LIN {X 0,Y 285.275,Z 343.324,A -85,B 0,C 180,E1 -18502.278,E2 -18502.278} C_VEL
LIN {X 0,Y 279.28,Z 333.872,A -85,B 0,C 180,E1 -18504.288,E2 -18504.288} C_VEL
LIN {X 0,Y 273.466,Z 325.227,A -85,B 0,C 180,E1 -18506.402,E2 -18506.402} C_VEL
LIN {X 0,Y 268.524,Z 318.8,A -85,B 0,C 180,E1 -18508.326,E2 -18508.326} C_VEL
LIN {X 0,Y 265.812,Z 315.625,A -85,B 0,C 180,E1 -18509.442,E2 -18509.442} C_VEL
LIN {X 0,Y 264.728,Z 313.915,A -85,B 0,C 180,E1 -18509.928,E2 -18509.928} C_VEL
LIN {X 0,Y 262.153,Z 311.495,A -85,B 0,C 180,E1 -18511.038,E2 -18511.038} C_VEL
LIN {X 0,Y 260.63,Z 308.609,A -85,B 0,C 180,E1 -18511.807,E2 -18511.807} C_VEL
LIN {X 0,Y 258.077,Z 306.933,A -85,B 0,C 180,E1 -18512.972,E2 -18512.972} C_VEL
LIN {X 0,Y 256.551,Z 304.575,A -85,B 0,C 180,E1 -18513.786,E2 -18513.786} C_VEL
LIN {X 0,Y 256.134,Z 302.894,A -85,B 0,C 180,E1 -18514.093,E2 -18514.093} C_VEL
LIN {X 0,Y 256.099,Z 302.893,A -85,B 0,C 180,E1 -18517.407,E2 -18517.407} C_VEL
LIN {X 0,Y 256.184,Z 302.852,A -85,B 0,C 180,E1 -18520.78,E2 -18520.78} C_VEL
LIN {X 0,Y 256.293,Z 302.86,A -85,B 0,C 180,E1 -18524.085,E2 -18524.085} C_VEL
LIN {X 0,Y 256.292,Z 302.834,A -85,B 0,C 180,E1 -18527.328,E2 -18527.328} C_VEL
LIN {X 0,Y 256.514,Z 302.81,A -85,B 0,C 180,E1 -18532.127,E2 -18532.127} C_VEL
LIN {X 0,Y 256.498,Z 302.847,A -85,B 0,C 180,E1 -18536.859,E2 -18536.859} C_VEL
LIN {X 0,Y 256.756,Z 302.772,A -85,B 0,C 180,E1 -18540,E2 -18540} C_VEL
LIN {X 0,Y 256.497,Z 302.827,A -85,B 0,C 180,E1 -18543.142,E2 -18543.142} C_VEL
LIN {X 0,Y 256.514,Z 302.799,A -85,B 0,C 180,E1 -18547.874,E2 -18547.874} C_VEL
LIN {X 0,Y 256.293,Z 302.863,A -85,B 0,C 180,E1 -18552.672,E2 -18552.672} C_VEL
LIN {X 0,Y 256.26,Z 302.84,A -85,B 0,C 180,E1 -18556.286,E2 -18556.286} C_VEL
LIN {X 0,Y 256.162,Z 302.855,A -85,B 0,C 180,E1 -18560.896,E2 -18560.896} C_VEL
LIN {X 0,Y 256.17,Z 302.889,A -85,B 0,C 180,E1 -18565.13,E2 -18565.13} C_VEL
LIN {X 0,Y 256.122,Z 302.89,A -85,B 0,C 180,E1 -18566.371,E2 -18566.371} C_VEL
LIN {X 0,Y 256.849,Z 305.157,A -85,B 0,C 180,E1 -18566.839,E2 -18566.839} C_VEL
LIN {X 0,Y 258.629,Z 307.429,A -85,B 0,C 180,E1 -18567.75,E2 -18567.75} C_VEL
LIN {X 0,Y 260.674,Z 308.807,A -85,B 0,C 180,E1 -18568.678,E2 -18568.678} C_VEL
LIN {X 0,Y 262.404,Z 311.878,A -85,B 0,C 180,E1 -18569.537,E2 -18569.537} C_VEL
LIN {X 0,Y 265.164,Z 314.465,A -85,B 0,C 180,E1 -18570.717,E2 -18570.717} C_VEL
LIN {X 0,Y 267.552,Z 317.88,A -85,B 0,C 180,E1 -18571.748,E2 -18571.748} C_VEL
LIN {X 0,Y 269.408,Z 319.837,A -85,B 0,C 180,E1 -18572.481,E2 -18572.481} C_VEL
LIN {X 0,Y 272.405,Z 323.638,A -85,B 0,C 180,E1 -18573.645,E2 -18573.645} C_VEL
LIN {X 0,Y 277.071,Z 329.846,A -85,B 0,C 180,E1 -18575.356,E2 -18575.356} C_VEL
LIN {X 0,Y 282.926,Z 337.789,A -85,B 0,C 180,E1 -18577.336,E2 -18577.336} C_VEL
LIN {X 0,Y 289.288,Z 347.193,A -85,B 0,C 180,E1 -18579.335,E2 -18579.335} C_VEL
LIN {X 0,Y 297.565,Z 360.153,A -85,B 0,C 180,E1 -18581.721,E2 -18581.721} C_VEL
LIN {X 0,Y 305.62,Z 374.188,A -85,B 0,C 180,E1 -18583.871,E2 -18583.871} C_VEL
LIN {X 0,Y 306.514,Z 376.066,A -85,B 0,C 180,E1 -18584.108,E2 -18584.108} C_VEL
LIN {X 0,Y 299.995,Z 497.473,A -85,B 0,C 180,E1 -18586.903,E2 -18586.903} C_VEL
LIN {X 0,Y 298.313,Z 513.582,A -85,B 0,C 180,E1 -18587.48,E2 -18587.48} C_VEL
LIN {X 0,Y 296.185,Z 528.781,A -85,B 0,C 180,E1 -18588.251,E2 -18588.251} C_VEL
LIN {X 0,Y 293.455,Z 544.075,A -85,B 0,C 180,E1 -18589.261,E2 -18589.261} C_VEL
LIN {X 0,Y 290.548,Z 557.266,A -85,B 0,C 180,E1 -18590.359,E2 -18590.359} C_VEL
LIN {X 0,Y 286.959,Z 571.758,A -85,B 0,C 180,E1 -18591.848,E2 -18591.848} C_VEL
LIN {X 0,Y 282.878,Z 585.913,A -85,B 0,C 180,E1 -18593.618,E2 -18593.618} C_VEL
LIN {X 0,Y 278.715,Z 599.171,A -85,B 0,C 180,E1 -18595.653,E2 -18595.653} C_VEL
LIN {X 0,Y 274.546,Z 611.271,A -85,B 0,C 180,E1 -18597.916,E2 -18597.916} C_VEL
LIN {X 0,Y 270.52,Z 622.375,A -85,B 0,C 180,E1 -18600.422,E2 -18600.422} C_VEL
LIN {X 0,Y 266.38,Z 633.115,A -85,B 0,C 180,E1 -18603.352,E2 -18603.352} C_VEL
LIN {X 0,Y 263.033,Z 642.124,A -85,B 0,C 180,E1 -18606.373,E2 -18606.373} C_VEL
LIN {X 0,Y 260.17,Z 649.651,A -85,B 0,C 180,E1 -18609.441,E2 -18609.441} C_VEL
LIN {X 0,Y 257.502,Z 657.205,A -85,B 0,C 180,E1 -18613.347,E2 -18613.347} C_VEL
LIN {X 0,Y 255.967,Z 661.885,A -85,B 0,C 180,E1 -18616.504,E2 -18616.504} C_VEL
LIN {X 0,Y 255.175,Z 664.727,A -85,B 0,C 180,E1 -18618.884,E2 -18618.884} C_VEL
LIN {X 0,Y 254.496,Z 667.617,A -85,B 0,C 180,E1 -18622.063,E2 -18622.063} C_VEL
LIN {X 0,Y 254.141,Z 669.513,A -85,B 0,C 180,E1 -18625.241,E2 -18625.241} C_VEL
LIN {X 0,Y 254.078,Z 670.469,A -85,B 0,C 180,E1 -18628.415,E2 -18628.415} C_VEL
LIN {X 0,Y 254.078,Z 670.481,A -85,B 0,C 180,E1 -18631.585,E2 -18631.585} C_VEL
LIN {X 0,Y 254.141,Z 669.574,A -85,B 0,C 180,E1 -18634.759,E2 -18634.759} C_VEL
LIN {X 0,Y 254.494,Z 667.702,A -85,B 0,C 180,E1 -18637.936,E2 -18637.936} C_VEL
LIN {X 0,Y 255.145,Z 664.86,A -85,B 0,C 180,E1 -18641.117,E2 -18641.117} C_VEL
LIN {X 0,Y 256.293,Z 660.99,A -85,B 0,C 180,E1 -18644.288,E2 -18644.288} C_VEL
LIN {X 0,Y 258.026,Z 655.765,A -85,B 0,C 180,E1 -18647.576,E2 -18647.576} C_VEL
LIN {X 0,Y 260.127,Z 649.916,A -85,B 0,C 180,E1 -18650.562,E2 -18650.562} C_VEL
LIN {X 0,Y 263.41,Z 641.424,A -85,B 0,C 180,E1 -18654.009,E2 -18654.009} C_VEL
LIN {X 0,Y 266.775,Z 632.258,A -85,B 0,C 180,E1 -18657.029,E2 -18657.029} C_VEL
LIN {X 0,Y 270.404,Z 622.812,A -85,B 0,C 180,E1 -18659.592,E2 -18659.592} C_VEL
LIN {X 0,Y 274.457,Z 611.863,A -85,B 0,C 180,E1 -18662.079,E2 -18662.079} C_VEL
LIN {X 0,Y 278.265,Z 600.716,A -85,B 0,C 180,E1 -18664.191,E2 -18664.191} C_VEL
LIN {X 0,Y 282.046,Z 588.931,A -85,B 0,C 180,E1 -18666.063,E2 -18666.063} C_VEL
LIN {X 0,Y 285.784,Z 576.531,A -85,B 0,C 180,E1 -18667.714,E2 -18667.714} C_VEL
LIN {X 0,Y 289.199,Z 563.238,A -85,B 0,C 180,E1 -18669.186,E2 -18669.186} C_VEL
LIN {X 0,Y 292.454,Z 549.191,A -85,B 0,C 180,E1 -18670.454,E2 -18670.454} C_VEL
LIN {X 0,Y 295.442,Z 534.168,A -85,B 0,C 180,E1 -18671.536,E2 -18671.536} C_VEL
LIN {X 0,Y 297.702,Z 518.897,A -85,B 0,C 180,E1 -18672.398,E2 -18672.398} C_VEL
LIN {X 0,Y 299.684,Z 502.058,A -85,B 0,C 180,E1 -18673.063,E2 -18673.063} C_VEL
LIN {X 0,Y 301.058,Z 481.051,A -85,B 0,C 180,E1 -18673.617,E2 -18673.617} C_VEL
LIN {X 0,Y 306.585,Z 376.776,A -85,B 0,C 180,E1 -18675.989,E2 -18675.989} C_VEL
LIN {X 0,Y 306.295,Z 375.437,A -85,B 0,C 180,E1 -18676.09,E2 -18676.09} C_VEL
LIN {X 0,Y 299.197,Z 362.765,A -85,B 0,C 180,E1 -18677.975,E2 -18677.975} C_VEL
LIN {X 0,Y 291.683,Z 350.766,A -85,B 0,C 180,E1 -18680.102,E2 -18680.102} C_VEL
LIN {X 0,Y 287.132,Z 343.847,A -85,B 0,C 180,E1 -18681.48,E2 -18681.48} C_VEL
LIN {X 0,Y 284.356,Z 340.758,A -85,B 0,C 180,E1 -18682.318,E2 -18682.318} C_VEL
LIN {X 0,Y 279.14,Z 337.36,A -85,B 0,C 180,E1 -18683.882,E2 -18683.882} C_VEL
LIN {X 0,Y 273.02,Z 333.547,A -85,B 0,C 180,E1 -18685.87,E2 -18685.87} C_VEL
LIN {X 0,Y 271.247,Z 331.735,A -85,B 0,C 180,E1 -18686.516,E2 -18686.516} C_VEL
LIN {X 0,Y 269.262,Z 329.124,A -85,B 0,C 180,E1 -18687.291,E2 -18687.291} C_VEL
LIN {X 0,Y 265.972,Z 324.859,A -85,B 0,C 180,E1 -18688.637,E2 -18688.637} C_VEL
LIN {X 0,Y 263.083,Z 321.248,A -85,B 0,C 180,E1 -18689.886,E2 -18689.886} C_VEL
LIN {X 0,Y 262.021,Z 319.981,A -85,B 0,C 180,E1 -18690.361,E2 -18690.361} C_VEL
LIN {X 0,Y 259.368,Z 316.979,A -85,B 0,C 180,E1 -18691.587,E2 -18691.587} C_VEL
LIN {X 0,Y 258.32,Z 315.094,A -85,B 0,C 180,E1 -18692.134,E2 -18692.134} C_VEL
LIN {X 0,Y 255.6,Z 312.813,A -85,B 0,C 180,E1 -18693.46,E2 -18693.46} C_VEL
LIN {X 0,Y 253.93,Z 309.833,A -85,B 0,C 180,E1 -18694.423,E2 -18694.423} C_VEL
LIN {X 0,Y 250.638,Z 307.386,A -85,B 0,C 180,E1 -18696.229,E2 -18696.229} C_VEL
LIN {X 0,Y 249.411,Z 305.23,A -85,B 0,C 180,E1 -18697.039,E2 -18697.039} C_VEL
LIN {X 0,Y 249.069,Z 303.741,A -85,B 0,C 180,E1 -18697.39,E2 -18697.39} C_VEL
LIN {X 0,Y 249.135,Z 303.748,A -85,B 0,C 180,E1 -18701.922,E2 -18701.922} C_VEL
LIN {X 0,Y 249.196,Z 303.728,A -85,B 0,C 180,E1 -18705.296,E2 -18705.296} C_VEL
LIN {X 0,Y 249.423,Z 303.689,A -85,B 0,C 180,E1 -18710.465,E2 -18710.465} C_VEL
LIN {X 0,Y 249.46,Z 303.724,A -85,B 0,C 180,E1 -18713.529,E2 -18713.529} C_VEL
LIN {X 0,Y 249.674,Z 303.664,A -85,B 0,C 180,E1 -18718.387,E2 -18718.387} C_VEL
LIN {X 0,Y 249.674,Z 303.684,A -85,B 0,C 180,E1 -18721.613,E2 -18721.613} C_VEL
LIN {X 0,Y 249.46,Z 303.713,A -85,B 0,C 180,E1 -18726.47,E2 -18726.47} C_VEL
LIN {X 0,Y 249.387,Z 303.699,A -85,B 0,C 180,E1 -18729.734,E2 -18729.734} C_VEL
LIN {X 0,Y 249.204,Z 303.75,A -85,B 0,C 180,E1 -18734.703,E2 -18734.703} C_VEL
LIN {X 0,Y 249.138,Z 303.758,A -85,B 0,C 180,E1 -18738.077,E2 -18738.077} C_VEL
LIN {X 0,Y 249.053,Z 303.773,A -85,B 0,C 180,E1 -18742.283,E2 -18742.283} C_VEL
LIN {X 0,Y 249.862,Z 306.296,A -85,B 0,C 180,E1 -18742.916,E2 -18742.916} C_VEL
LIN {X 0,Y 251.817,Z 308.516,A -85,B 0,C 180,E1 -18744.09,E2 -18744.09} C_VEL
LIN {X 0,Y 253.91,Z 309.796,A -85,B 0,C 180,E1 -18745.199,E2 -18745.199} C_VEL
LIN {X 0,Y 255.481,Z 312.696,A -85,B 0,C 180,E1 -18746.113,E2 -18746.113} C_VEL
LIN {X 0,Y 258.017,Z 314.954,A -85,B 0,C 180,E1 -18747.364,E2 -18747.364} C_VEL
LIN {X 0,Y 258.576,Z 315.522,A -85,B 0,C 180,E1 -18747.634,E2 -18747.634} C_VEL
LIN {X 0,Y 260.685,Z 318.703,A -85,B 0,C 180,E1 -18748.678,E2 -18748.678} C_VEL
LIN {X 0,Y 262.953,Z 321.044,A -85,B 0,C 180,E1 -18749.688,E2 -18749.688} C_VEL
LIN {X 0,Y 265.557,Z 324.493,A -85,B 0,C 180,E1 -18750.83,E2 -18750.83} C_VEL
LIN {X 0,Y 267.011,Z 326.216,A -85,B 0,C 180,E1 -18751.432,E2 -18751.432} C_VEL
LIN {X 0,Y 271.996,Z 332.99,A -85,B 0,C 180,E1 -18753.417,E2 -18753.417} C_VEL
LIN {X 0,Y 278.858,Z 343.518,A -85,B 0,C 180,E1 -18755.936,E2 -18755.936} C_VEL
LIN {X 0,Y 286.061,Z 355.576,A -85,B 0,C 180,E1 -18758.347,E2 -18758.347} C_VEL
LIN {X 0,Y 293.093,Z 368.397,A -85,B 0,C 180,E1 -18760.517,E2 -18760.517} C_VEL
LIN {X 0,Y 299.812,Z 382.28,A -85,B 0,C 180,E1 -18762.471,E2 -18762.471} C_VEL
LIN {X 0,Y 301.353,Z 385.582,A -85,B 0,C 180,E1 -18762.901,E2 -18762.901} C_VEL
LIN {X 0,Y 294.372,Z 510.514,A -85,B 0,C 180,E1 -18765.799,E2 -18765.799} C_VEL
LIN {X 0,Y 292.365,Z 527.573,A -85,B 0,C 180,E1 -18766.402,E2 -18766.402} C_VEL
LIN {X 0,Y 289.707,Z 543.728,A -85,B 0,C 180,E1 -18767.215,E2 -18767.215} C_VEL
LIN {X 0,Y 286.53,Z 559.561,A -85,B 0,C 180,E1 -18768.294,E2 -18768.294} C_VEL
LIN {X 0,Y 283.015,Z 574.179,A -85,B 0,C 180,E1 -18769.553,E2 -18769.553} C_VEL
LIN {X 0,Y 278.905,Z 588.943,A -85,B 0,C 180,E1 -18771.143,E2 -18771.143} C_VEL
LIN {X 0,Y 274.506,Z 602.929,A -85,B 0,C 180,E1 -18773.012,E2 -18773.012} C_VEL
LIN {X 0,Y 270.049,Z 615.655,A -85,B 0,C 180,E1 -18775.072,E2 -18775.072} C_VEL
LIN {X 0,Y 265.467,Z 628.288,A -85,B 0,C 180,E1 -18777.582,E2 -18777.582} C_VEL
LIN {X 0,Y 261.478,Z 639.066,A -85,B 0,C 180,E1 -18780.183,E2 -18780.183} C_VEL
LIN {X 0,Y 257.372,Z 649.469,A -85,B 0,C 180,E1 -18783.221,E2 -18783.221} C_VEL
LIN {X 0,Y 254.04,Z 658.16,A -85,B 0,C 180,E1 -18786.351,E2 -18786.351} C_VEL
LIN {X 0,Y 251.411,Z 665.441,A -85,B 0,C 180,E1 -18789.548,E2 -18789.548} C_VEL
LIN {X 0,Y 249.437,Z 671.625,A -85,B 0,C 180,E1 -18792.877,E2 -18792.877} C_VEL
LIN {X 0,Y 247.855,Z 677.362,A -85,B 0,C 180,E1 -18796.889,E2 -18796.889} C_VEL
LIN {X 0,Y 247.105,Z 680.799,A -85,B 0,C 180,E1 -18800.175,E2 -18800.175} C_VEL
LIN {X 0,Y 246.858,Z 683.304,A -85,B 0,C 180,E1 -18803.461,E2 -18803.461} C_VEL
LIN {X 0,Y 246.852,Z 684.721,A -85,B 0,C 180,E1 -18806.736,E2 -18806.736} C_VEL
LIN {X 0,Y 246.981,Z 685.254,A -85,B 0,C 180,E1 -18810,E2 -18810} C_VEL
LIN {X 0,Y 246.852,Z 684.711,A -85,B 0,C 180,E1 -18813.264,E2 -18813.264} C_VEL
LIN {X 0,Y 246.859,Z 683.284,A -85,B 0,C 180,E1 -18816.539,E2 -18816.539} C_VEL
LIN {X 0,Y 247.105,Z 680.77,A -85,B 0,C 180,E1 -18819.825,E2 -18819.825} C_VEL
LIN {X 0,Y 248.115,Z 676.241,A -85,B 0,C 180,E1 -18823.932,E2 -18823.932} C_VEL
LIN {X 0,Y 249.436,Z 671.576,A -85,B 0,C 180,E1 -18827.124,E2 -18827.124} C_VEL
LIN {X 0,Y 252.01,Z 663.718,A -85,B 0,C 180,E1 -18831.256,E2 -18831.256} C_VEL
LIN {X 0,Y 254.904,Z 655.834,A -85,B 0,C 180,E1 -18834.517,E2 -18834.517} C_VEL
LIN {X 0,Y 258.342,Z 646.883,A -85,B 0,C 180,E1 -18837.547,E2 -18837.547} C_VEL
LIN {X 0,Y 262.56,Z 635.997,A -85,B 0,C 180,E1 -18840.569,E2 -18840.569} C_VEL
LIN {X 0,Y 266.111,Z 626.507,A -85,B 0,C 180,E1 -18842.779,E2 -18842.779} C_VEL
LIN {X 0,Y 270.039,Z 615.479,A -85,B 0,C 180,E1 -18844.929,E2 -18844.929} C_VEL
LIN {X 0,Y 274.491,Z 602.717,A -85,B 0,C 180,E1 -18846.991,E2 -18846.991} C_VEL
LIN {X 0,Y 278.509,Z 589.956,A -85,B 0,C 180,E1 -18848.709,E2 -18848.709} C_VEL
LIN {X 0,Y 282.572,Z 575.469,A -85,B 0,C 180,E1 -18850.29,E2 -18850.29} C_VEL
LIN {X 0,Y 286.078,Z 561.175,A -85,B 0,C 180,E1 -18851.552,E2 -18851.552} C_VEL
LIN {X 0,Y 289.237,Z 545.847,A -85,B 0,C 180,E1 -18852.634,E2 -18852.634} C_VEL
LIN {X 0,Y 292.012,Z 529.58,A -85,B 0,C 180,E1 -18853.486,E2 -18853.486} C_VEL
LIN {X 0,Y 294.055,Z 512.875,A -85,B 0,C 180,E1 -18854.098,E2 -18854.098} C_VEL
LIN {X 0,Y 295.614,Z 486.575,A -85,B 0,C 180,E1 -18854.773,E2 -18854.773} C_VEL
LIN {X 0,Y 301.244,Z 385.521,A -85,B 0,C 180,E1 -18857.076,E2 -18857.076} C_VEL
LIN {X 0,Y 294.208,Z 370.745,A -85,B 0,C 180,E1 -18859.093,E2 -18859.093} C_VEL
LIN {X 0,Y 287.651,Z 358.497,A -85,B 0,C 180,E1 -18861.084,E2 -18861.084} C_VEL
LIN {X 0,Y 280.685,Z 346.559,A -85,B 0,C 180,E1 -18863.361,E2 -18863.361} C_VEL
LIN {X 0,Y 275.917,Z 339.051,A -85,B 0,C 180,E1 -18865.033,E2 -18865.033} C_VEL
LIN {X 0,Y 270.151,Z 330.37,A -85,B 0,C 180,E1 -18867.219,E2 -18867.219} C_VEL
LIN {X 0,Y 265.908,Z 324.844,A -85,B 0,C 180,E1 -18868.934,E2 -18868.934} C_VEL
LIN {X 0,Y 263.062,Z 321.269,A -85,B 0,C 180,E1 -18870.16,E2 -18870.16} C_VEL
LIN {X 0,Y 261.902,Z 319.861,A -85,B 0,C 180,E1 -18870.678,E2 -18870.678} C_VEL
LIN {X 0,Y 259.328,Z 316.934,A -85,B 0,C 180,E1 -18871.864,E2 -18871.864} C_VEL
LIN {X 0,Y 258.206,Z 315.058,A -85,B 0,C 180,E1 -18872.438,E2 -18872.438} C_VEL
LIN {X 0,Y 255.549,Z 312.778,A -85,B 0,C 180,E1 -18873.73,E2 -18873.73} C_VEL
LIN {X 0,Y 253.879,Z 309.778,A -85,B 0,C 180,E1 -18874.689,E2 -18874.689} C_VEL
LIN {X 0,Y 250.643,Z 307.395,A -85,B 0,C 180,E1 -18876.449,E2 -18876.449} C_VEL
LIN {X 0,Y 249.403,Z 305.259,A -85,B 0,C 180,E1 -18877.258,E2 -18877.258} C_VEL
LIN {X 0,Y 249.052,Z 303.764,A -85,B 0,C 180,E1 -18877.607,E2 -18877.607} C_VEL
LIN {X 0,Y 249.138,Z 303.743,A -85,B 0,C 180,E1 -18881.923,E2 -18881.923} C_VEL
LIN {X 0,Y 249.199,Z 303.721,A -85,B 0,C 180,E1 -18885.297,E2 -18885.297} C_VEL
LIN {X 0,Y 249.386,Z 303.729,A -85,B 0,C 180,E1 -18890.517,E2 -18890.517} C_VEL
LIN {X 0,Y 249.452,Z 303.679,A -85,B 0,C 180,E1 -18893.53,E2 -18893.53} C_VEL
LIN {X 0,Y 249.675,Z 303.678,A -85,B 0,C 180,E1 -18898.387,E2 -18898.387} C_VEL
LIN {X 0,Y 249.674,Z 303.653,A -85,B 0,C 180,E1 -18901.613,E2 -18901.613} C_VEL
LIN {X 0,Y 249.44,Z 303.689,A -85,B 0,C 180,E1 -18906.711,E2 -18906.711} C_VEL
LIN {X 0,Y 249.342,Z 303.703,A -85,B 0,C 180,E1 -18909.737,E2 -18909.737} C_VEL
LIN {X 0,Y 249.196,Z 303.715,A -85,B 0,C 180,E1 -18914.704,E2 -18914.704} C_VEL
LIN {X 0,Y 249.135,Z 303.759,A -85,B 0,C 180,E1 -18918.078,E2 -18918.078} C_VEL
LIN {X 0,Y 249.037,Z 303.739,A -85,B 0,C 180,E1 -18922.395,E2 -18922.395} C_VEL
LIN {X 0,Y 249.035,Z 303.765,A -85,B 0,C 180,E1 -18922.888,E2 -18922.888} C_VEL
LIN {X 0,Y 249.722,Z 306.013,A -85,B 0,C 180,E1 -18923.424,E2 -18923.424} C_VEL
LIN {X 0,Y 251.586,Z 308.326,A -85,B 0,C 180,E1 -18924.553,E2 -18924.553} C_VEL
LIN {X 0,Y 253.921,Z 309.828,A -85,B 0,C 180,E1 -18925.79,E2 -18925.79} C_VEL
LIN {X 0,Y 255.614,Z 312.839,A -85,B 0,C 180,E1 -18926.758,E2 -18926.758} C_VEL
LIN {X 0,Y 258.488,Z 315.485,A -85,B 0,C 180,E1 -18928.161,E2 -18928.161} C_VEL
LIN {X 0,Y 260.8,Z 318.863,A -85,B 0,C 180,E1 -18929.293,E2 -18929.293} C_VEL
LIN {X 0,Y 262.853,Z 320.924,A -85,B 0,C 180,E1 -18930.199,E2 -18930.199} C_VEL
LIN {X 0,Y 265.628,Z 324.576,A -85,B 0,C 180,E1 -18931.408,E2 -18931.408} C_VEL
LIN {X 0,Y 267.03,Z 326.203,A -85,B 0,C 180,E1 -18931.984,E2 -18931.984} C_VEL
LIN {X 0,Y 270.974,Z 331.365,A -85,B 0,C 180,E1 -18933.551,E2 -18933.551} C_VEL
LIN {X 0,Y 277.003,Z 339.459,A -85,B 0,C 180,E1 -18935.758,E2 -18935.758} C_VEL
LIN {X 0,Y 284.758,Z 350.731,A -85,B 0,C 180,E1 -18938.342,E2 -18938.342} C_VEL
LIN {X 0,Y 293.587,Z 364.766,A -85,B 0,C 180,E1 -18941.005,E2 -18941.005} C_VEL
LIN {X 0,Y 301.429,Z 378.591,A -85,B 0,C 180,E1 -18943.18,E2 -18943.18} C_VEL
LIN {X 0,Y 294.933,Z 496.966,A -85,B 0,C 180,E1 -18945.947,E2 -18945.947} C_VEL
LIN {X 0,Y 293.248,Z 512.887,A -85,B 0,C 180,E1 -18946.507,E2 -18946.507} C_VEL
LIN {X 0,Y 290.915,Z 528.997,A -85,B 0,C 180,E1 -18947.317,E2 -18947.317} C_VEL
LIN {X 0,Y 288.115,Z 544.289,A -85,B 0,C 180,E1 -18948.34,E2 -18948.34} C_VEL
LIN {X 0,Y 285.105,Z 557.479,A -85,B 0,C 180,E1 -18949.447,E2 -18949.447} C_VEL
LIN {X 0,Y 281.748,Z 570.559,A -85,B 0,C 180,E1 -18950.782,E2 -18950.782} C_VEL
LIN {X 0,Y 277.6,Z 584.956,A -85,B 0,C 180,E1 -18952.584,E2 -18952.584} C_VEL
LIN {X 0,Y 273.574,Z 597.276,A -85,B 0,C 180,E1 -18954.463,E2 -18954.463} C_VEL
LIN {X 0,Y 269.106,Z 609.715,A -85,B 0,C 180,E1 -18956.74,E2 -18956.74} C_VEL
LIN {X 0,Y 264.892,Z 621.112,A -85,B 0,C 180,E1 -18959.288,E2 -18959.288} C_VEL
LIN {X 0,Y 260.996,Z 630.875,A -85,B 0,C 180,E1 -18961.886,E2 -18961.886} C_VEL
LIN {X 0,Y 257.317,Z 640.237,A -85,B 0,C 180,E1 -18964.954,E2 -18964.954} C_VEL
LIN {X 0,Y 254.161,Z 648.073,A -85,B 0,C 180,E1 -18968.081,E2 -18968.081} C_VEL
LIN {X 0,Y 251.668,Z 654.605,A -85,B 0,C 180,E1 -18971.268,E2 -18971.268} C_VEL
LIN {X 0,Y 249.772,Z 659.884,A -85,B 0,C 180,E1 -18974.496,E2 -18974.496} C_VEL
LIN {X 0,Y 248.656,Z 663.146,A -85,B 0,C 180,E1 -18976.932,E2 -18976.932} C_VEL
LIN {X 0,Y 247.763,Z 666.493,A -85,B 0,C 180,E1 -18980.201,E2 -18980.201} C_VEL
LIN {X 0,Y 247.196,Z 668.926,A -85,B 0,C 180,E1 -18983.47,E2 -18983.47} C_VEL
LIN {X 0,Y 247.015,Z 670.301,A -85,B 0,C 180,E1 -18986.738,E2 -18986.738} C_VEL
LIN {X 0,Y 246.99,Z 670.831,A -85,B 0,C 180,E1 -18990,E2 -18990} C_VEL
LIN {X 0,Y 247.014,Z 670.338,A -85,B 0,C 180,E1 -18993.262,E2 -18993.262} C_VEL
LIN {X 0,Y 247.195,Z 668.997,A -85,B 0,C 180,E1 -18996.53,E2 -18996.53} C_VEL
LIN {X 0,Y 247.755,Z 666.601,A -85,B 0,C 180,E1 -18999.799,E2 -18999.799} C_VEL
LIN {X 0,Y 248.626,Z 663.298,A -85,B 0,C 180,E1 -19003.07,E2 -19003.07} C_VEL
LIN {X 0,Y 250.608,Z 657.647,A -85,B 0,C 180,E1 -19007.101,E2 -19007.101} C_VEL
LIN {X 0,Y 253.413,Z 650.124,A -85,B 0,C 180,E1 -19011.133,E2 -19011.133} C_VEL
LIN {X 0,Y 256.874,Z 641.632,A -85,B 0,C 180,E1 -19014.66,E2 -19014.66} C_VEL
LIN {X 0,Y 260.406,Z 632.465,A -85,B 0,C 180,E1 -19017.746,E2 -19017.746} C_VEL
LIN {X 0,Y 264.196,Z 623.019,A -85,B 0,C 180,E1 -19020.359,E2 -19020.359} C_VEL
LIN {X 0,Y 268.123,Z 612.898,A -85,B 0,C 180,E1 -19022.719,E2 -19022.719} C_VEL
LIN {X 0,Y 272.379,Z 600.922,A -85,B 0,C 180,E1 -19025.036,E2 -19025.036} C_VEL
LIN {X 0,Y 276.343,Z 589.134,A -85,B 0,C 180,E1 -19026.929,E2 -19026.929} C_VEL
LIN {X 0,Y 280.173,Z 576.735,A -85,B 0,C 180,E1 -19028.607,E2 -19028.607} C_VEL
LIN {X 0,Y 283.72,Z 563.441,A -85,B 0,C 180,E1 -19030.093,E2 -19030.093} C_VEL
LIN {X 0,Y 287.104,Z 549.391,A -85,B 0,C 180,E1 -19031.37,E2 -19031.37} C_VEL
LIN {X 0,Y 290.16,Z 534.367,A -85,B 0,C 180,E1 -19032.466,E2 -19032.466} C_VEL
LIN {X 0,Y 292.513,Z 519.094,A -85,B 0,C 180,E1 -19033.334,E2 -19033.334} C_VEL
LIN {X 0,Y 294.523,Z 502.501,A -85,B 0,C 180,E1 -19033.996,E2 -19033.996} C_VEL
LIN {X 0,Y 295.987,Z 480.767,A -85,B 0,C 180,E1 -19034.575,E2 -19034.575} C_VEL
LIN {X 0,Y 301.593,Z 379.214,A -85,B 0,C 180,E1 -19036.903,E2 -19036.903} C_VEL
LIN {X 0,Y 300.741,Z 377.174,A -85,B 0,C 180,E1 -19037.148,E2 -19037.148} C_VEL
LIN {X 0,Y 292.638,Z 363.121,A -85,B 0,C 180,E1 -19039.417,E2 -19039.417} C_VEL
LIN {X 0,Y 283.622,Z 348.999,A -85,B 0,C 180,E1 -19042.176,E2 -19042.176} C_VEL
LIN {X 0,Y 276.328,Z 338.452,A -85,B 0,C 180,E1 -19044.647,E2 -19044.647} C_VEL
LIN {X 0,Y 271.247,Z 331.735,A -85,B 0,C 180,E1 -19046.516,E2 -19046.516} C_VEL
LIN {X 0,Y 268.561,Z 329.352,A -85,B 0,C 180,E1 -19047.515,E2 -19047.515} C_VEL
LIN {X 0,Y 263.721,Z 327.214,A -85,B 0,C 180,E1 -19049.331,E2 -19049.331} C_VEL
LIN {X 0,Y 259.146,Z 325.104,A -85,B 0,C 180,E1 -19051.214,E2 -19051.214} C_VEL
LIN {X 0,Y 256.843,Z 322.762,A -85,B 0,C 180,E1 -19052.31,E2 -19052.31} C_VEL
LIN {X 0,Y 255.802,Z 321.309,A -85,B 0,C 180,E1 -19052.849,E2 -19052.849} C_VEL
LIN {X 0,Y 253.145,Z 318.616,A -85,B 0,C 180,E1 -19054.229,E2 -19054.229} C_VEL
LIN {X 0,Y 251.679,Z 316.151,A -85,B 0,C 180,E1 -19055.099,E2 -19055.099} C_VEL
LIN {X 0,Y 248.857,Z 313.93,A -85,B 0,C 180,E1 -19056.71,E2 -19056.71} C_VEL
LIN {X 0,Y 247.239,Z 311.109,A -85,B 0,C 180,E1 -19057.819,E2 -19057.819} C_VEL
LIN {X 0,Y 246.9,Z 310.49,A -85,B 0,C 180,E1 -19058.062,E2 -19058.062} C_VEL
LIN {X 0,Y 244.122,Z 308.824,A -85,B 0,C 180,E1 -19059.899,E2 -19059.899} C_VEL
LIN {X 0,Y 242.516,Z 306.416,A -85,B 0,C 180,E1 -19061.192,E2 -19061.192} C_VEL
LIN {X 0,Y 242.074,Z 304.631,A -85,B 0,C 180,E1 -19061.705,E2 -19061.705} C_VEL
LIN {X 0,Y 242.155,Z 304.6,A -85,B 0,C 180,E1 -19064.858,E2 -19064.858} C_VEL
LIN {X 0,Y 242.364,Z 304.568,A -85,B 0,C 180,E1 -19070.371,E2 -19070.371} C_VEL
LIN {X 0,Y 242.432,Z 304.596,A -85,B 0,C 180,E1 -19073.341,E2 -19073.341} C_VEL
LIN {X 0,Y 242.634,Z 304.539,A -85,B 0,C 180,E1 -19078.34,E2 -19078.34} C_VEL
LIN {X 0,Y 242.635,Z 304.558,A -85,B 0,C 180,E1 -19081.66,E2 -19081.66} C_VEL
LIN {X 0,Y 242.432,Z 304.592,A -85,B 0,C 180,E1 -19086.659,E2 -19086.659} C_VEL
LIN {X 0,Y 242.313,Z 304.578,A -85,B 0,C 180,E1 -19090.022,E2 -19090.022} C_VEL
LIN {X 0,Y 242.165,Z 304.625,A -85,B 0,C 180,E1 -19095.141,E2 -19095.141} C_VEL
LIN {X 0,Y 242.129,Z 304.78,A -85,B 0,C 180,E1 -19098.017,E2 -19098.017} C_VEL
LIN {X 0,Y 242.727,Z 306.822,A -85,B 0,C 180,E1 -19098.626,E2 -19098.626} C_VEL
LIN {X 0,Y 244.301,Z 308.998,A -85,B 0,C 180,E1 -19099.866,E2 -19099.866} C_VEL
LIN {X 0,Y 247.087,Z 310.745,A -85,B 0,C 180,E1 -19101.701,E2 -19101.701} C_VEL
LIN {X 0,Y 248.601,Z 313.641,A -85,B 0,C 180,E1 -19102.764,E2 -19102.764} C_VEL
LIN {X 0,Y 251.002,Z 315.788,A -85,B 0,C 180,E1 -19104.173,E2 -19104.173} C_VEL
LIN {X 0,Y 251.924,Z 316.542,A -85,B 0,C 180,E1 -19104.682,E2 -19104.682} C_VEL
LIN {X 0,Y 254.097,Z 319.804,A -85,B 0,C 180,E1 -19105.925,E2 -19105.925} C_VEL
LIN {X 0,Y 256.437,Z 322.017,A -85,B 0,C 180,E1 -19107.105,E2 -19107.105} C_VEL
LIN {X 0,Y 259.001,Z 325.572,A -85,B 0,C 180,E1 -19108.387,E2 -19108.387} C_VEL
LIN {X 0,Y 260.555,Z 327.248,A -85,B 0,C 180,E1 -19109.101,E2 -19109.101} C_VEL
LIN {X 0,Y 263.742,Z 331.281,A -85,B 0,C 180,E1 -19110.525,E2 -19110.525} C_VEL
LIN {X 0,Y 269.115,Z 338.679,A -85,B 0,C 180,E1 -19112.756,E2 -19112.756} C_VEL
LIN {X 0,Y 275.643,Z 348.883,A -85,B 0,C 180,E1 -19115.247,E2 -19115.247} C_VEL
LIN {X 0,Y 282.45,Z 360.484,A -85,B 0,C 180,E1 -19117.618,E2 -19117.618} C_VEL
LIN {X 0,Y 289.599,Z 373.783,A -85,B 0,C 180,E1 -19119.91,E2 -19119.91} C_VEL
LIN {X 0,Y 296.012,Z 387.458,A -85,B 0,C 180,E1 -19121.85,E2 -19121.85} C_VEL
LIN {X 0,Y 296.357,Z 388.202,A -85,B 0,C 180,E1 -19121.951,E2 -19121.951} C_VEL
LIN {X 0,Y 292.743,Z 450.63,A -85,B 0,C 180,E1 -19123.385,E2 -19123.385} C_VEL
LIN {X 0,Y 289.263,Z 510.944,A -85,B 0,C 180,E1 -19124.836,E2 -19124.836} C_VEL
LIN {X 0,Y 287.134,Z 528.294,A -85,B 0,C 180,E1 -19125.461,E2 -19125.461} C_VEL
LIN {X 0,Y 284.524,Z 543.528,A -85,B 0,C 180,E1 -19126.242,E2 -19126.242} C_VEL
LIN {X 0,Y 281.248,Z 559.359,A -85,B 0,C 180,E1 -19127.327,E2 -19127.327} C_VEL
LIN {X 0,Y 277.611,Z 573.975,A -85,B 0,C 180,E1 -19128.595,E2 -19128.595} C_VEL
LIN {X 0,Y 273.298,Z 588.988,A -85,B 0,C 180,E1 -19130.232,E2 -19130.232} C_VEL
LIN {X 0,Y 268.828,Z 602.724,A -85,B 0,C 180,E1 -19132.095,E2 -19132.095} C_VEL
LIN {X 0,Y 264.196,Z 615.448,A -85,B 0,C 180,E1 -19134.181,E2 -19134.181} C_VEL
LIN {X 0,Y 259.431,Z 628.081,A -85,B 0,C 180,E1 -19136.731,E2 -19136.731} C_VEL
LIN {X 0,Y 255.26,Z 638.858,A -85,B 0,C 180,E1 -19139.379,E2 -19139.379} C_VEL
LIN {X 0,Y 250.966,Z 649.261,A -85,B 0,C 180,E1 -19142.48,E2 -19142.48} C_VEL
LIN {X 0,Y 247.354,Z 658.157,A -85,B 0,C 180,E1 -19145.762,E2 -19145.762} C_VEL
LIN {X 0,Y 244.67,Z 665.232,A -85,B 0,C 180,E1 -19148.958,E2 -19148.958} C_VEL
LIN {X 0,Y 242.582,Z 671.282,A -85,B 0,C 180,E1 -19152.29,E2 -19152.29} C_VEL
LIN {X 0,Y 240.874,Z 677.154,A -85,B 0,C 180,E1 -19156.502,E2 -19156.502} C_VEL
LIN {X 0,Y 240.041,Z 680.59,A -85,B 0,C 180,E1 -19159.883,E2 -19159.883} C_VEL
LIN {X 0,Y 239.77,Z 683.096,A -85,B 0,C 180,E1 -19163.267,E2 -19163.267} C_VEL
LIN {X 0,Y 239.758,Z 684.513,A -85,B 0,C 180,E1 -19166.639,E2 -19166.639} C_VEL
LIN {X 0,Y 239.89,Z 685.047,A -85,B 0,C 180,E1 -19170,E2 -19170} C_VEL
LIN {X 0,Y 239.758,Z 684.503,A -85,B 0,C 180,E1 -19173.361,E2 -19173.361} C_VEL
LIN {X 0,Y 239.77,Z 683.075,A -85,B 0,C 180,E1 -19176.733,E2 -19176.733} C_VEL
LIN {X 0,Y 240.041,Z 680.56,A -85,B 0,C 180,E1 -19180.118,E2 -19180.118} C_VEL
LIN {X 0,Y 240.87,Z 677.113,A -85,B 0,C 180,E1 -19183.498,E2 -19183.498} C_VEL
LIN {X 0,Y 242.58,Z 671.228,A -85,B 0,C 180,E1 -19187.71,E2 -19187.71} C_VEL
LIN {X 0,Y 245.315,Z 663.506,A -85,B 0,C 180,E1 -19191.866,E2 -19191.866} C_VEL
LIN {X 0,Y 248.718,Z 654.809,A -85,B 0,C 180,E1 -19195.526,E2 -19195.526} C_VEL
LIN {X 0,Y 252.493,Z 645.429,A -85,B 0,C 180,E1 -19198.695,E2 -19198.695} C_VEL
LIN {X 0,Y 256.372,Z 635.784,A -85,B 0,C 180,E1 -19201.389,E2 -19201.389} C_VEL
LIN {X 0,Y 260.087,Z 626.294,A -85,B 0,C 180,E1 -19203.638,E2 -19203.638} C_VEL
LIN {X 0,Y 264.193,Z 615.267,A -85,B 0,C 180,E1 -19205.82,E2 -19205.82} C_VEL
LIN {X 0,Y 268.41,Z 603.682,A -85,B 0,C 180,E1 -19207.737,E2 -19207.737} C_VEL
LIN {X 0,Y 272.476,Z 591.235,A -85,B 0,C 180,E1 -19209.457,E2 -19209.457} C_VEL
LIN {X 0,Y 276.706,Z 576.843,A -85,B 0,C 180,E1 -19211.086,E2 -19211.086} C_VEL
LIN {X 0,Y 280.797,Z 560.962,A -85,B 0,C 180,E1 -19212.514,E2 -19212.514} C_VEL
LIN {X 0,Y 284.043,Z 545.632,A -85,B 0,C 180,E1 -19213.606,E2 -19213.606} C_VEL
LIN {X 0,Y 286.884,Z 529.503,A -85,B 0,C 180,E1 -19214.454,E2 -19214.454} C_VEL
LIN {X 0,Y 288.897,Z 513.718,A -85,B 0,C 180,E1 -19215.04,E2 -19215.04} C_VEL
LIN {X 0,Y 290.337,Z 491.726,A -85,B 0,C 180,E1 -19215.629,E2 -19215.629} C_VEL
LIN {X 0,Y 296.242,Z 388.038,A -85,B 0,C 180,E1 -19218.029,E2 -19218.029} C_VEL
LIN {X 0,Y 290.005,Z 374.852,A -85,B 0,C 180,E1 -19219.899,E2 -19219.899} C_VEL
LIN {X 0,Y 284.038,Z 363.501,A -85,B 0,C 180,E1 -19221.788,E2 -19221.788} C_VEL
LIN {X 0,Y 277.217,Z 351.602,A -85,B 0,C 180,E1 -19224.11,E2 -19224.11} C_VEL
LIN {X 0,Y 272.617,Z 344.24,A -85,B 0,C 180,E1 -19225.791,E2 -19225.791} C_VEL
LIN {X 0,Y 267.307,Z 336.079,A -85,B 0,C 180,E1 -19227.887,E2 -19227.887} C_VEL
LIN {X 0,Y 263.17,Z 330.698,A -85,B 0,C 180,E1 -19229.621,E2 -19229.621} C_VEL
LIN {X 0,Y 259.674,Z 326.214,A -85,B 0,C 180,E1 -19231.2,E2 -19231.2} C_VEL
LIN {X 0,Y 256.854,Z 322.782,A -85,B 0,C 180,E1 -19232.557,E2 -19232.557} C_VEL
LIN {X 0,Y 255.89,Z 321.413,A -85,B 0,C 180,E1 -19233.053,E2 -19233.053} C_VEL
LIN {X 0,Y 253.035,Z 318.509,A -85,B 0,C 180,E1 -19234.526,E2 -19234.526} C_VEL
LIN {X 0,Y 251.656,Z 316.12,A -85,B 0,C 180,E1 -19235.345,E2 -19235.345} C_VEL
LIN {X 0,Y 248.853,Z 313.937,A -85,B 0,C 180,E1 -19236.931,E2 -19236.931} C_VEL
LIN {X 0,Y 247.218,Z 311.132,A -85,B 0,C 180,E1 -19238.037,E2 -19238.037} C_VEL
LIN {X 0,Y 246.878,Z 310.5,A -85,B 0,C 180,E1 -19238.28,E2 -19238.28} C_VEL
LIN {X 0,Y 244.083,Z 308.752,A -85,B 0,C 180,E1 -19240.116,E2 -19240.116} C_VEL
LIN {X 0,Y 242.581,Z 306.518,A -85,B 0,C 180,E1 -19241.307,E2 -19241.307} C_VEL
LIN {X 0,Y 242.089,Z 304.619,A -85,B 0,C 180,E1 -19241.87,E2 -19241.87} C_VEL
LIN {X 0,Y 242.162,Z 304.602,A -85,B 0,C 180,E1 -19244.859,E2 -19244.859} C_VEL
LIN {X 0,Y 242.332,Z 304.609,A -85,B 0,C 180,E1 -19250.417,E2 -19250.417} C_VEL
LIN {X 0,Y 242.423,Z 304.554,A -85,B 0,C 180,E1 -19253.341,E2 -19253.341} C_VEL
LIN {X 0,Y 242.635,Z 304.555,A -85,B 0,C 180,E1 -19258.34,E2 -19258.34} C_VEL
LIN {X 0,Y 242.635,Z 304.529,A -85,B 0,C 180,E1 -19261.66,E2 -19261.66} C_VEL
LIN {X 0,Y 242.421,Z 304.563,A -85,B 0,C 180,E1 -19266.683,E2 -19266.683} C_VEL
LIN {X 0,Y 242.267,Z 304.588,A -85,B 0,C 180,E1 -19270.024,E2 -19270.024} C_VEL
LIN {X 0,Y 242.155,Z 304.59,A -85,B 0,C 180,E1 -19275.142,E2 -19275.142} C_VEL
LIN {X 0,Y 242.068,Z 304.703,A -85,B 0,C 180,E1 -19278.625,E2 -19278.625} C_VEL
LIN {X 0,Y 242.734,Z 306.858,A -85,B 0,C 180,E1 -19279.284,E2 -19279.284} C_VEL
LIN {X 0,Y 244.608,Z 309.256,A -85,B 0,C 180,E1 -19280.715,E2 -19280.715} C_VEL
LIN {X 0,Y 247.074,Z 310.739,A -85,B 0,C 180,E1 -19282.307,E2 -19282.307} C_VEL
LIN {X 0,Y 248.53,Z 313.527,A -85,B 0,C 180,E1 -19283.322,E2 -19283.322} C_VEL
LIN {X 0,Y 251.112,Z 315.836,A -85,B 0,C 180,E1 -19284.823,E2 -19284.823} C_VEL
LIN {X 0,Y 251.958,Z 316.596,A -85,B 0,C 180,E1 -19285.29,E2 -19285.29} C_VEL
LIN {X 0,Y 254.069,Z 319.795,A -85,B 0,C 180,E1 -19286.49,E2 -19286.49} C_VEL
LIN {X 0,Y 256.315,Z 321.918,A -85,B 0,C 180,E1 -19287.617,E2 -19287.617} C_VEL
LIN {X 0,Y 258.941,Z 325.542,A -85,B 0,C 180,E1 -19288.924,E2 -19288.924} C_VEL
LIN {X 0,Y 260.641,Z 327.384,A -85,B 0,C 180,E1 -19289.701,E2 -19289.701} C_VEL
LIN {X 0,Y 263.719,Z 331.266,A -85,B 0,C 180,E1 -19291.066,E2 -19291.066} C_VEL
LIN {X 0,Y 268.333,Z 337.385,A -85,B 0,C 180,E1 -19292.976,E2 -19292.976} C_VEL
LIN {X 0,Y 274.339,Z 345.624,A -85,B 0,C 180,E1 -19295.248,E2 -19295.248} C_VEL
LIN {X 0,Y 281.492,Z 356.217,A -85,B 0,C 180,E1 -19297.712,E2 -19297.712} C_VEL
LIN {X 0,Y 290.206,Z 370.316,A -85,B 0,C 180,E1 -19300.434,E2 -19300.434} C_VEL
LIN {X 0,Y 296.496,Z 381.547,A -85,B 0,C 180,E1 -19302.251,E2 -19302.251} C_VEL
LIN {X 0,Y 289.919,Z 496.681,A -85,B 0,C 180,E1 -19304.96,E2 -19304.96} C_VEL
LIN {X 0,Y 288.139,Z 513.106,A -85,B 0,C 180,E1 -19305.535,E2 -19305.535} C_VEL
LIN {X 0,Y 285.746,Z 529.213,A -85,B 0,C 180,E1 -19306.354,E2 -19306.354} C_VEL
LIN {X 0,Y 282.861,Z 544.503,A -85,B 0,C 180,E1 -19307.386,E2 -19307.386} C_VEL
LIN {X 0,Y 279.748,Z 557.693,A -85,B 0,C 180,E1 -19308.501,E2 -19308.501} C_VEL
LIN {X 0,Y 276.099,Z 571.372,A -85,B 0,C 180,E1 -19309.92,E2 -19309.92} C_VEL
LIN {X 0,Y 271.983,Z 585.167,A -85,B 0,C 180,E1 -19311.673,E2 -19311.673} C_VEL
LIN {X 0,Y 268.176,Z 596.424,A -85,B 0,C 180,E1 -19313.402,E2 -19313.402} C_VEL
LIN {X 0,Y 263.787,Z 608.334,A -85,B 0,C 180,E1 -19315.564,E2 -19315.564} C_VEL
LIN {X 0,Y 259.35,Z 619.85,A -85,B 0,C 180,E1 -19318.101,E2 -19318.101} C_VEL
LIN {X 0,Y 254.722,Z 631.086,A -85,B 0,C 180,E1 -19321.129,E2 -19321.129} C_VEL
LIN {X 0,Y 250.833,Z 640.449,A -85,B 0,C 180,E1 -19324.26,E2 -19324.26} C_VEL
LIN {X 0,Y 247.512,Z 648.284,A -85,B 0,C 180,E1 -19327.46,E2 -19327.46} C_VEL
LIN {X 0,Y 244.9,Z 654.815,A -85,B 0,C 180,E1 -19330.73,E2 -19330.73} C_VEL
LIN {X 0,Y 242.886,Z 660.094,A -85,B 0,C 180,E1 -19334.045,E2 -19334.045} C_VEL
LIN {X 0,Y 241.699,Z 663.356,A -85,B 0,C 180,E1 -19336.549,E2 -19336.549} C_VEL
LIN {X 0,Y 240.722,Z 666.702,A -85,B 0,C 180,E1 -19339.911,E2 -19339.911} C_VEL
LIN {X 0,Y 240.134,Z 669.134,A -85,B 0,C 180,E1 -19343.277,E2 -19343.277} C_VEL
LIN {X 0,Y 239.917,Z 670.509,A -85,B 0,C 180,E1 -19346.641,E2 -19346.641} C_VEL
LIN {X 0,Y 239.921,Z 671.037,A -85,B 0,C 180,E1 -19350,E2 -19350} C_VEL
LIN {X 0,Y 239.916,Z 670.545,A -85,B 0,C 180,E1 -19353.359,E2 -19353.359} C_VEL
LIN {X 0,Y 240.134,Z 669.205,A -85,B 0,C 180,E1 -19356.723,E2 -19356.723} C_VEL
LIN {X 0,Y 240.713,Z 666.809,A -85,B 0,C 180,E1 -19360.089,E2 -19360.089} C_VEL
LIN {X 0,Y 241.666,Z 663.506,A -85,B 0,C 180,E1 -19363.453,E2 -19363.453} C_VEL
LIN {X 0,Y 243.271,Z 659.048,A -85,B 0,C 180,E1 -19366.792,E2 -19366.792} C_VEL
LIN {X 0,Y 245.453,Z 653.527,A -85,B 0,C 180,E1 -19370.096,E2 -19370.096} C_VEL
LIN {X 0,Y 248.221,Z 646.759,A -85,B 0,C 180,E1 -19373.352,E2 -19373.352} C_VEL
LIN {X 0,Y 251.671,Z 638.56,A -85,B 0,C 180,E1 -19376.539,E2 -19376.539} C_VEL
LIN {X 0,Y 255.745,Z 628.794,A -85,B 0,C 180,E1 -19379.646,E2 -19379.646} C_VEL
LIN {X 0,Y 259.857,Z 618.745,A -85,B 0,C 180,E1 -19382.286,E2 -19382.286} C_VEL
LIN {X 0,Y 264.44,Z 606.897,A -85,B 0,C 180,E1 -19384.848,E2 -19384.848} C_VEL
LIN {X 0,Y 269.084,Z 593.85,A -85,B 0,C 180,E1 -19387.155,E2 -19387.155} C_VEL
LIN {X 0,Y 273.455,Z 580.807,A -85,B 0,C 180,E1 -19389.025,E2 -19389.025} C_VEL
LIN {X 0,Y 277.554,Z 566.516,A -85,B 0,C 180,E1 -19390.736,E2 -19390.736} C_VEL
LIN {X 0,Y 281.357,Z 551.572,A -85,B 0,C 180,E1 -19392.168,E2 -19392.168} C_VEL
LIN {X 0,Y 284.739,Z 535.753,A -85,B 0,C 180,E1 -19393.351,E2 -19393.351} C_VEL
LIN {X 0,Y 287.269,Z 520.052,A -85,B 0,C 180,E1 -19394.267,E2 -19394.267} C_VEL
LIN {X 0,Y 289.437,Z 502.966,A -85,B 0,C 180,E1 -19394.962,E2 -19394.962} C_VEL
LIN {X 0,Y 290.961,Z 481.418,A -85,B 0,C 180,E1 -19395.542,E2 -19395.542} C_VEL
LIN {X 0,Y 296.629,Z 381.672,A -85,B 0,C 180,E1 -19397.857,E2 -19397.857} C_VEL
LIN {X 0,Y 288.846,Z 367.969,A -85,B 0,C 180,E1 -19400.123,E2 -19400.123} C_VEL
LIN {X 0,Y 280.247,Z 354.263,A -85,B 0,C 180,E1 -19402.86,E2 -19402.86} C_VEL
LIN {X 0,Y 273.037,Z 343.75,A -85,B 0,C 180,E1 -19405.397,E2 -19405.397} C_VEL
LIN {X 0,Y 267.011,Z 335.56,A -85,B 0,C 180,E1 -19407.736,E2 -19407.736} C_VEL
LIN {X 0,Y 263.178,Z 330.676,A -85,B 0,C 180,E1 -19409.349,E2 -19409.349} C_VEL
LIN {X 0,Y 259.838,Z 326.365,A -85,B 0,C 180,E1 -19410.866,E2 -19410.866} C_VEL
LIN {X 0,Y 257.016,Z 323.05,A -85,B 0,C 180,E1 -19412.219,E2 -19412.219} C_VEL
LIN {X 0,Y 256.843,Z 322.762,A -85,B 0,C 180,E1 -19412.31,E2 -19412.31} C_VEL
LIN {X 0,Y 254.67,Z 320.446,A -85,B 0,C 180,E1 -19413.408,E2 -19413.408} C_VEL
LIN {X 0,Y 252.321,Z 319.135,A -85,B 0,C 180,E1 -19414.588,E2 -19414.588} C_VEL
LIN {X 0,Y 244.765,Z 317.064,A -85,B 0,C 180,E1 -19418.817,E2 -19418.817} C_VEL
LIN {X 0,Y 242.221,Z 315.09,A -85,B 0,C 180,E1 -19420.618,E2 -19420.618} C_VEL
LIN {X 0,Y 240.598,Z 312.27,A -85,B 0,C 180,E1 -19422.029,E2 -19422.029} C_VEL
LIN {X 0,Y 240.292,Z 311.479,A -85,B 0,C 180,E1 -19422.335,E2 -19422.335} C_VEL
LIN {X 0,Y 237.312,Z 309.782,A -85,B 0,C 180,E1 -19424.981,E2 -19424.981} C_VEL
LIN {X 0,Y 235.68,Z 307.543,A -85,B 0,C 180,E1 -19426.857,E2 -19426.857} C_VEL
LIN {X 0,Y 235.124,Z 305.501,A -85,B 0,C 180,E1 -19427.813,E2 -19427.813} C_VEL
LIN {X 0,Y 235.376,Z 305.442,A -85,B 0,C 180,E1 -19431.414,E2 -19431.414} C_VEL
LIN {X 0,Y 235.403,Z 305.466,A -85,B 0,C 180,E1 -19433.141,E2 -19433.141} C_VEL
LIN {X 0,Y 235.594,Z 305.415,A -85,B 0,C 180,E1 -19438.29,E2 -19438.29} C_VEL
LIN {X 0,Y 235.594,Z 305.433,A -85,B 0,C 180,E1 -19441.709,E2 -19441.709} C_VEL
LIN {X 0,Y 235.403,Z 305.471,A -85,B 0,C 180,E1 -19446.858,E2 -19446.858} C_VEL
LIN {X 0,Y 235.237,Z 305.457,A -85,B 0,C 180,E1 -19450.326,E2 -19450.326} C_VEL
LIN {X 0,Y 235.144,Z 305.519,A -85,B 0,C 180,E1 -19451.912,E2 -19451.912} C_VEL
LIN {X 0,Y 235.705,Z 307.602,A -85,B 0,C 180,E1 -19452.812,E2 -19452.812} C_VEL
LIN {X 0,Y 237.446,Z 309.918,A -85,B 0,C 180,E1 -19454.79,E2 -19454.79} C_VEL
LIN {X 0,Y 240.438,Z 311.727,A -85,B 0,C 180,E1 -19457.434,E2 -19457.434} C_VEL
LIN {X 0,Y 241.761,Z 314.516,A -85,B 0,C 180,E1 -19458.649,E2 -19458.649} C_VEL
LIN {X 0,Y 244.239,Z 316.815,A -85,B 0,C 180,E1 -19460.474,E2 -19460.474} C_VEL
LIN {X 0,Y 245.382,Z 317.648,A -85,B 0,C 180,E1 -19461.236,E2 -19461.236} C_VEL
LIN {X 0,Y 247.135,Z 320.563,A -85,B 0,C 180,E1 -19462.466,E2 -19462.466} C_VEL
LIN {X 0,Y 249.997,Z 323.151,A -85,B 0,C 180,E1 -19464.166,E2 -19464.166} C_VEL
LIN {X 0,Y 252.493,Z 326.659,A -85,B 0,C 180,E1 -19465.614,E2 -19465.614} C_VEL
LIN {X 0,Y 254.414,Z 328.634,A -85,B 0,C 180,E1 -19466.617,E2 -19466.617} C_VEL
LIN {X 0,Y 257.324,Z 332.398,A -85,B 0,C 180,E1 -19468.091,E2 -19468.091} C_VEL
LIN {X 0,Y 259.092,Z 334.776,A -85,B 0,C 180,E1 -19468.942,E2 -19468.942} C_VEL
LIN {X 0,Y 262.283,Z 338.789,A -85,B 0,C 180,E1 -19470.382,E2 -19470.382} C_VEL
LIN {X 0,Y 266.474,Z 344.727,A -85,B 0,C 180,E1 -19472.169,E2 -19472.169} C_VEL
LIN {X 0,Y 272.635,Z 354.541,A -85,B 0,C 180,E1 -19474.605,E2 -19474.605} C_VEL
LIN {X 0,Y 279.004,Z 365.673,A -85,B 0,C 180,E1 -19476.914,E2 -19476.914} C_VEL
LIN {X 0,Y 285.797,Z 378.566,A -85,B 0,C 180,E1 -19479.182,E2 -19479.182} C_VEL
LIN {X 0,Y 291.448,Z 390.73,A -85,B 0,C 180,E1 -19480.965,E2 -19480.965} C_VEL
LIN {X 0,Y 289.545,Z 424.085,A -85,B 0,C 180,E1 -19481.76,E2 -19481.76} C_VEL
LIN {X 0,Y 284.361,Z 510.108,A -85,B 0,C 180,E1 -19483.802,E2 -19483.802} C_VEL
LIN {X 0,Y 282.222,Z 527.417,A -85,B 0,C 180,E1 -19484.424,E2 -19484.424} C_VEL
LIN {X 0,Y 279.428,Z 543.329,A -85,B 0,C 180,E1 -19485.233,E2 -19485.233} C_VEL
LIN {X 0,Y 276.031,Z 559.156,A -85,B 0,C 180,E1 -19486.321,E2 -19486.321} C_VEL
LIN {X 0,Y 272.3,Z 573.772,A -85,B 0,C 180,E1 -19487.602,E2 -19487.602} C_VEL
LIN {X 0,Y 267.835,Z 588.779,A -85,B 0,C 180,E1 -19489.251,E2 -19489.251} C_VEL
LIN {X 0,Y 263.219,Z 602.518,A -85,B 0,C 180,E1 -19491.138,E2 -19491.138} C_VEL
LIN {X 0,Y 258.403,Z 615.241,A -85,B 0,C 180,E1 -19493.249,E2 -19493.249} C_VEL
LIN {X 0,Y 253.45,Z 627.873,A -85,B 0,C 180,E1 -19495.839,E2 -19495.839} C_VEL
LIN {X 0,Y 249.083,Z 638.649,A -85,B 0,C 180,E1 -19498.535,E2 -19498.535} C_VEL
LIN {X 0,Y 244.577,Z 649.052,A -85,B 0,C 180,E1 -19501.697,E2 -19501.697} C_VEL
LIN {X 0,Y 240.693,Z 658.214,A -85,B 0,C 180,E1 -19505.166,E2 -19505.166} C_VEL
LIN {X 0,Y 237.948,Z 665.022,A -85,B 0,C 180,E1 -19508.334,E2 -19508.334} C_VEL
LIN {X 0,Y 235.712,Z 671.072,A -85,B 0,C 180,E1 -19511.756,E2 -19511.756} C_VEL
LIN {X 0,Y 233.903,Z 676.945,A -85,B 0,C 180,E1 -19516.092,E2 -19516.092} C_VEL
LIN {X 0,Y 232.994,Z 680.382,A -85,B 0,C 180,E1 -19519.573,E2 -19519.573} C_VEL
LIN {X 0,Y 232.673,Z 682.888,A -85,B 0,C 180,E1 -19523.061,E2 -19523.061} C_VEL
LIN {X 0,Y 232.668,Z 684.306,A -85,B 0,C 180,E1 -19526.537,E2 -19526.537} C_VEL
LIN {X 0,Y 232.8,Z 684.84,A -85,B 0,C 180,E1 -19530,E2 -19530} C_VEL
LIN {X 0,Y 232.668,Z 684.296,A -85,B 0,C 180,E1 -19533.464,E2 -19533.464} C_VEL
LIN {X 0,Y 232.673,Z 682.866,A -85,B 0,C 180,E1 -19536.94,E2 -19536.94} C_VEL
LIN {X 0,Y 232.994,Z 680.35,A -85,B 0,C 180,E1 -19540.427,E2 -19540.427} C_VEL
LIN {X 0,Y 233.899,Z 676.903,A -85,B 0,C 180,E1 -19543.909,E2 -19543.909} C_VEL
LIN {X 0,Y 235.711,Z 671.017,A -85,B 0,C 180,E1 -19548.244,E2 -19548.244} C_VEL
LIN {X 0,Y 238.646,Z 663.294,A -85,B 0,C 180,E1 -19552.51,E2 -19552.51} C_VEL
LIN {X 0,Y 242.233,Z 654.597,A -85,B 0,C 180,E1 -19556.26,E2 -19556.26} C_VEL
LIN {X 0,Y 246.178,Z 645.216,A -85,B 0,C 180,E1 -19559.502,E2 -19559.502} C_VEL
LIN {X 0,Y 250.229,Z 635.571,A -85,B 0,C 180,E1 -19562.251,E2 -19562.251} C_VEL
LIN {X 0,Y 254.806,Z 624.339,A -85,B 0,C 180,E1 -19564.912,E2 -19564.912} C_VEL
LIN {X 0,Y 259.539,Z 612.112,A -85,B 0,C 180,E1 -19567.292,E2 -19567.292} C_VEL
LIN {X 0,Y 264.389,Z 598.754,A -85,B 0,C 180,E1 -19569.393,E2 -19569.393} C_VEL
LIN {X 0,Y 269.146,Z 584.221,A -85,B 0,C 180,E1 -19571.249,E2 -19571.249} C_VEL
LIN {X 0,Y 273.226,Z 569.994,A -85,B 0,C 180,E1 -19572.72,E2 -19572.72} C_VEL
LIN {X 0,Y 277.024,Z 554.654,A -85,B 0,C 180,E1 -19573.986,E2 -19573.986} C_VEL
LIN {X 0,Y 280.148,Z 539.035,A -85,B 0,C 180,E1 -19574.989,E2 -19574.989} C_VEL
LIN {X 0,Y 282.761,Z 522.684,A -85,B 0,C 180,E1 -19575.743,E2 -19575.743} C_VEL
LIN {X 0,Y 284.586,Z 505.513,A -85,B 0,C 180,E1 -19576.295,E2 -19576.295} C_VEL
LIN {X 0,Y 291.333,Z 390.656,A -85,B 0,C 180,E1 -19579.009,E2 -19579.009} C_VEL
LIN {X 0,Y 285.876,Z 378.95,A -85,B 0,C 180,E1 -19580.725,E2 -19580.725} C_VEL
LIN {X 0,Y 280.215,Z 368.042,A -85,B 0,C 180,E1 -19582.597,E2 -19582.597} C_VEL
LIN {X 0,Y 274.102,Z 357.11,A -85,B 0,C 180,E1 -19584.768,E2 -19584.768} C_VEL
LIN {X 0,Y 269.694,Z 349.945,A -85,B 0,C 180,E1 -19586.439,E2 -19586.439} C_VEL
LIN {X 0,Y 264.305,Z 341.496,A -85,B 0,C 180,E1 -19588.654,E2 -19588.654} C_VEL
LIN {X 0,Y 260.742,Z 336.85,A -85,B 0,C 180,E1 -19590.201,E2 -19590.201} C_VEL
LIN {X 0,Y 257.318,Z 332.404,A -85,B 0,C 180,E1 -19591.802,E2 -19591.802} C_VEL
LIN {X 0,Y 254.313,Z 328.514,A -85,B 0,C 180,E1 -19593.316,E2 -19593.316} C_VEL
LIN {X 0,Y 250.648,Z 324.324,A -85,B 0,C 180,E1 -19595.294,E2 -19595.294} C_VEL
LIN {X 0,Y 249.644,Z 322.662,A -85,B 0,C 180,E1 -19595.908,E2 -19595.908} C_VEL
LIN {X 0,Y 246.932,Z 320.29,A -85,B 0,C 180,E1 -19597.515,E2 -19597.515} C_VEL
LIN {X 0,Y 245.128,Z 317.241,A -85,B 0,C 180,E1 -19598.783,E2 -19598.783} C_VEL
LIN {X 0,Y 242.432,Z 315.291,A -85,B 0,C 180,E1 -19600.636,E2 -19600.636} C_VEL
LIN {X 0,Y 240.747,Z 312.661,A -85,B 0,C 180,E1 -19602.041,E2 -19602.041} C_VEL
LIN {X 0,Y 240.212,Z 311.451,A -85,B 0,C 180,E1 -19602.549,E2 -19602.549} C_VEL
LIN {X 0,Y 237.409,Z 309.882,A -85,B 0,C 180,E1 -19604.988,E2 -19604.988} C_VEL
LIN {X 0,Y 235.645,Z 307.444,A -85,B 0,C 180,E1 -19606.965,E2 -19606.965} C_VEL
LIN {X 0,Y 235.12,Z 305.473,A -85,B 0,C 180,E1 -19607.813,E2 -19607.813} C_VEL
LIN {X 0,Y 235.33,Z 305.456,A -85,B 0,C 180,E1 -19611.413,E2 -19611.413} C_VEL
LIN {X 0,Y 235.373,Z 305.432,A -85,B 0,C 180,E1 -19613.141,E2 -19613.141} C_VEL
LIN {X 0,Y 235.595,Z 305.431,A -85,B 0,C 180,E1 -19618.291,E2 -19618.291} C_VEL
LIN {X 0,Y 235.594,Z 305.405,A -85,B 0,C 180,E1 -19621.71,E2 -19621.71} C_VEL
LIN {X 0,Y 235.373,Z 305.438,A -85,B 0,C 180,E1 -19626.86,E2 -19626.86} C_VEL
LIN {X 0,Y 235.214,Z 305.471,A -85,B 0,C 180,E1 -19630.328,E2 -19630.328} C_VEL
LIN {X 0,Y 235.126,Z 305.535,A -85,B 0,C 180,E1 -19632.68,E2 -19632.68} C_VEL
LIN {X 0,Y 235.635,Z 307.405,A -85,B 0,C 180,E1 -19633.475,E2 -19633.475} C_VEL
LIN {X 0,Y 236.987,Z 309.464,A -85,B 0,C 180,E1 -19635.04,E2 -19635.04} C_VEL
LIN {X 0,Y 239.685,Z 311.29,A -85,B 0,C 180,E1 -19637.491,E2 -19637.491} C_VEL
LIN {X 0,Y 240.373,Z 311.627,A -85,B 0,C 180,E1 -19638.044,E2 -19638.044} C_VEL
LIN {X 0,Y 241.652,Z 314.342,A -85,B 0,C 180,E1 -19639.209,E2 -19639.209} C_VEL
LIN {X 0,Y 243.957,Z 316.597,A -85,B 0,C 180,E1 -19640.91,E2 -19640.91} C_VEL
LIN {X 0,Y 245.284,Z 317.493,A -85,B 0,C 180,E1 -19641.785,E2 -19641.785} C_VEL
LIN {X 0,Y 247.213,Z 320.637,A -85,B 0,C 180,E1 -19643.121,E2 -19643.121} C_VEL
LIN {X 0,Y 249.943,Z 323.047,A -85,B 0,C 180,E1 -19644.725,E2 -19644.725} C_VEL
LIN {X 0,Y 252.52,Z 326.695,A -85,B 0,C 180,E1 -19646.211,E2 -19646.211} C_VEL
LIN {X 0,Y 254.209,Z 328.375,A -85,B 0,C 180,E1 -19647.085,E2 -19647.085} C_VEL
LIN {X 0,Y 257.081,Z 332.196,A -85,B 0,C 180,E1 -19648.544,E2 -19648.544} C_VEL
LIN {X 0,Y 258.457,Z 333.847,A -85,B 0,C 180,E1 -19649.198,E2 -19649.198} C_VEL
LIN {X 0,Y 262.826,Z 339.561,A -85,B 0,C 180,E1 -19651.173,E2 -19651.173} C_VEL
LIN {X 0,Y 266.739,Z 344.804,A -85,B 0,C 180,E1 -19652.805,E2 -19652.805} C_VEL
LIN {X 0,Y 273.558,Z 354.5,A -85,B 0,C 180,E1 -19655.412,E2 -19655.412} C_VEL
LIN {X 0,Y 280.825,Z 365.859,A -85,B 0,C 180,E1 -19657.931,E2 -19657.931} C_VEL
LIN {X 0,Y 287.947,Z 377.838,A -85,B 0,C 180,E1 -19660.186,E2 -19660.186} C_VEL
LIN {X 0,Y 291.609,Z 384.464,A -85,B 0,C 180,E1 -19661.281,E2 -19661.281} C_VEL
LIN {X 0,Y 284.909,Z 497.369,A -85,B 0,C 180,E1 -19663.961,E2 -19663.961} C_VEL
LIN {X 0,Y 283.135,Z 513.325,A -85,B 0,C 180,E1 -19664.532,E2 -19664.532} C_VEL
LIN {X 0,Y 280.646,Z 529.429,A -85,B 0,C 180,E1 -19665.353,E2 -19665.353} C_VEL
LIN {X 0,Y 277.683,Z 544.716,A -85,B 0,C 180,E1 -19666.395,E2 -19666.395} C_VEL
LIN {X 0,Y 274.46,Z 557.906,A -85,B 0,C 180,E1 -19667.517,E2 -19667.517} C_VEL
LIN {X 0,Y 270.511,Z 572.198,A -85,B 0,C 180,E1 -19669.023,E2 -19669.023} C_VEL
LIN {X 0,Y 266.444,Z 585.379,A -85,B 0,C 180,E1 -19670.725,E2 -19670.725} C_VEL
LIN {X 0,Y 262.857,Z 595.574,A -85,B 0,C 180,E1 -19672.294,E2 -19672.294} C_VEL
LIN {X 0,Y 258.012,Z 608.367,A -85,B 0,C 180,E1 -19674.632,E2 -19674.632} C_VEL
LIN {X 0,Y 253.312,Z 620.062,A -85,B 0,C 180,E1 -19677.247,E2 -19677.247} C_VEL
LIN {X 0,Y 248.477,Z 631.297,A -85,B 0,C 180,E1 -19680.332,E2 -19680.332} C_VEL
LIN {X 0,Y 244.395,Z 640.66,A -85,B 0,C 180,E1 -19683.53,E2 -19683.53} C_VEL
LIN {X 0,Y 240.908,Z 648.495,A -85,B 0,C 180,E1 -19686.807,E2 -19686.807} C_VEL
LIN {X 0,Y 238.155,Z 655.026,A -85,B 0,C 180,E1 -19690.162,E2 -19690.162} C_VEL
LIN {X 0,Y 235.578,Z 661.464,A -85,B 0,C 180,E1 -19694.425,E2 -19694.425} C_VEL
LIN {X 0,Y 234.17,Z 665.355,A -85,B 0,C 180,E1 -19697.873,E2 -19697.873} C_VEL
LIN {X 0,Y 233.342,Z 668.242,A -85,B 0,C 180,E1 -19701.339,E2 -19701.339} C_VEL
LIN {X 0,Y 232.921,Z 670.135,A -85,B 0,C 180,E1 -19704.806,E2 -19704.806} C_VEL
LIN {X 0,Y 232.811,Z 671.09,A -85,B 0,C 180,E1 -19708.27,E2 -19708.27} C_VEL
LIN {X 0,Y 232.811,Z 671.102,A -85,B 0,C 180,E1 -19711.73,E2 -19711.73} C_VEL
LIN {X 0,Y 232.913,Z 670.156,A -85,B 0,C 180,E1 -19715.281,E2 -19715.281} C_VEL
LIN {X 0,Y 233.339,Z 668.325,A -85,B 0,C 180,E1 -19718.661,E2 -19718.661} C_VEL
LIN {X 0,Y 234.145,Z 665.484,A -85,B 0,C 180,E1 -19722.129,E2 -19722.129} C_VEL
LIN {X 0,Y 235.543,Z 661.615,A -85,B 0,C 180,E1 -19725.577,E2 -19725.577} C_VEL
LIN {X 0,Y 238.092,Z 655.229,A -85,B 0,C 180,E1 -19729.844,E2 -19729.844} C_VEL
LIN {X 0,Y 240.855,Z 648.755,A -85,B 0,C 180,E1 -19733.198,E2 -19733.198} C_VEL
LIN {X 0,Y 244.343,Z 640.979,A -85,B 0,C 180,E1 -19736.476,E2 -19736.476} C_VEL
LIN {X 0,Y 247.834,Z 632.878,A -85,B 0,C 180,E1 -19739.286,E2 -19739.286} C_VEL
LIN {X 0,Y 251.952,Z 623.432,A -85,B 0,C 180,E1 -19742.004,E2 -19742.004} C_VEL
LIN {X 0,Y 256.241,Z 613.177,A -85,B 0,C 180,E1 -19744.481,E2 -19744.481} C_VEL
LIN {X 0,Y 260.83,Z 601.331,A -85,B 0,C 180,E1 -19746.835,E2 -19746.835} C_VEL
LIN {X 0,Y 265.117,Z 589.542,A -85,B 0,C 180,E1 -19748.775,E2 -19748.775} C_VEL
LIN {X 0,Y 269.568,Z 575.735,A -85,B 0,C 180,E1 -19750.676,E2 -19750.676} C_VEL
LIN {X 0,Y 273.455,Z 562.269,A -85,B 0,C 180,E1 -19752.177,E2 -19752.177} C_VEL
LIN {X 0,Y 277.098,Z 547.811,A -85,B 0,C 180,E1 -19753.469,E2 -19753.469} C_VEL
LIN {X 0,Y 280.291,Z 532.171,A -85,B 0,C 180,E1 -19754.593,E2 -19754.593} C_VEL
LIN {X 0,Y 282.86,Z 516.269,A -85,B 0,C 180,E1 -19755.461,E2 -19755.461} C_VEL
LIN {X 0,Y 284.835,Z 499.342,A -85,B 0,C 180,E1 -19756.107,E2 -19756.107} C_VEL
LIN {X 0,Y 288.719,Z 435.1,A -85,B 0,C 180,E1 -19757.656,E2 -19757.656} C_VEL
LIN {X 0,Y 291.72,Z 384.564,A -85,B 0,C 180,E1 -19758.834,E2 -19758.834} C_VEL
LIN {X 0,Y 284.2,Z 371.292,A -85,B 0,C 180,E1 -19761.134,E2 -19761.134} C_VEL
LIN {X 0,Y 275.802,Z 357.768,A -85,B 0,C 180,E1 -19763.952,E2 -19763.952} C_VEL
LIN {X 0,Y 267.656,Z 345.912,A -85,B 0,C 180,E1 -19767.01,E2 -19767.01} C_VEL
LIN {X 0,Y 260.82,Z 336.877,A -85,B 0,C 180,E1 -19769.904,E2 -19769.904} C_VEL
LIN {X 0,Y 257.425,Z 332.509,A -85,B 0,C 180,E1 -19771.496,E2 -19771.496} C_VEL
LIN {X 0,Y 254.448,Z 328.701,A -85,B 0,C 180,E1 -19772.998,E2 -19772.998} C_VEL
LIN {X 0,Y 253.58,Z 327.647,A -85,B 0,C 180,E1 -19773.454,E2 -19773.454} C_VEL
LIN {X 0,Y 250.66,Z 324.273,A -85,B 0,C 180,E1 -19775.06,E2 -19775.06} C_VEL
LIN {X 0,Y 249.718,Z 322.733,A -85,B 0,C 180,E1 -19775.639,E2 -19775.639} C_VEL
LIN {X 0,Y 246.8,Z 320.094,A -85,B 0,C 180,E1 -19777.391,E2 -19777.391} C_VEL
LIN {X 0,Y 245.083,Z 317.218,A -85,B 0,C 180,E1 -19778.612,E2 -19778.612} C_VEL
LIN {X 0,Y 244.765,Z 317.064,A -85,B 0,C 180,E1 -19778.817,E2 -19778.817} C_VEL
LIN {X 0,Y 242.123,Z 316.379,A -85,B 0,C 180,E1 -19780.571,E2 -19780.571} C_VEL
LIN {X 0,Y 237.308,Z 316.709,A -85,B 0,C 180,E1 -19784.203,E2 -19784.203} C_VEL
LIN {X 0,Y 235.399,Z 315.931,A -85,B 0,C 180,E1 -19786.06,E2 -19786.06} C_VEL
LIN {X 0,Y 233.973,Z 313.121,A -85,B 0,C 180,E1 -19787.972,E2 -19787.972} C_VEL
LIN {X 0,Y 233.786,Z 312.455,A -85,B 0,C 180,E1 -19788.292,E2 -19788.292} C_VEL
LIN {X 0,Y 229.574,Z 309.284,A -85,B 0,C 180,E1 -19798.026,E2 -19798.026} C_VEL
LIN {X 0,Y 229.525,Z 309.09,A -85,B 0,C 180,E1 -19800.877,E2 -19800.877} C_VEL
LIN {X 0,Y 233.841,Z 312.602,A -85,B 0,C 180,E1 -19811.43,E2 -19811.43} C_VEL
LIN {X 0,Y 234.896,Z 315.191,A -85,B 0,C 180,E1 -19812.967,E2 -19812.967} C_VEL
LIN {X 0,Y 237.016,Z 317.435,A -85,B 0,C 180,E1 -19815.257,E2 -19815.257} C_VEL
LIN {X 0,Y 238.913,Z 318.552,A -85,B 0,C 180,E1 -19816.939,E2 -19816.939} C_VEL
LIN {X 0,Y 240.398,Z 321.391,A -85,B 0,C 180,E1 -19818.317,E2 -19818.317} C_VEL
LIN {X 0,Y 243.053,Z 323.781,A -85,B 0,C 180,E1 -19820.303,E2 -19820.303} C_VEL
LIN {X 0,Y 243.745,Z 324.504,A -85,B 0,C 180,E1 -19820.792,E2 -19820.792} C_VEL
LIN {X 0,Y 245.943,Z 327.724,A -85,B 0,C 180,E1 -19822.331,E2 -19822.331} C_VEL
LIN {X 0,Y 248.096,Z 329.698,A -85,B 0,C 180,E1 -19823.641,E2 -19823.641} C_VEL
LIN {X 0,Y 250.698,Z 333.269,A -85,B 0,C 180,E1 -19825.189,E2 -19825.189} C_VEL
LIN {X 0,Y 252.402,Z 335.165,A -85,B 0,C 180,E1 -19826.112,E2 -19826.112} C_VEL
LIN {X 0,Y 256.539,Z 340.576,A -85,B 0,C 180,E1 -19828.238,E2 -19828.238} C_VEL
LIN {X 0,Y 260.334,Z 345.635,A -85,B 0,C 180,E1 -19830.018,E2 -19830.018} C_VEL
LIN {X 0,Y 263.551,Z 350.232,A -85,B 0,C 180,E1 -19831.433,E2 -19831.433} C_VEL
LIN {X 0,Y 269.586,Z 360.105,A -85,B 0,C 180,E1 -19833.921,E2 -19833.921} C_VEL
LIN {X 0,Y 275.716,Z 371.028,A -85,B 0,C 180,E1 -19836.231,E2 -19836.231} C_VEL
LIN {X 0,Y 282.836,Z 384.895,A -85,B 0,C 180,E1 -19838.696,E2 -19838.696} C_VEL
LIN {X 0,Y 286.667,Z 393.36,A -85,B 0,C 180,E1 -19839.96,E2 -19839.96} C_VEL
LIN {X 0,Y 285.207,Z 418.275,A -85,B 0,C 180,E1 -19840.561,E2 -19840.561} C_VEL
LIN {X 0,Y 279.495,Z 509.918,A -85,B 0,C 180,E1 -19842.752,E2 -19842.752} C_VEL
LIN {X 0,Y 277.333,Z 527.035,A -85,B 0,C 180,E1 -19843.37,E2 -19843.37} C_VEL
LIN {X 0,Y 274.434,Z 543.129,A -85,B 0,C 180,E1 -19844.189,E2 -19844.189} C_VEL
LIN {X 0,Y 270.913,Z 558.954,A -85,B 0,C 180,E1 -19845.278,E2 -19845.278} C_VEL
LIN {X 0,Y 267.088,Z 573.569,A -85,B 0,C 180,E1 -19846.573,E2 -19846.573} C_VEL
LIN {X 0,Y 262.453,Z 588.589,A -85,B 0,C 180,E1 -19848.234,E2 -19848.234} C_VEL
LIN {X 0,Y 257.674,Z 602.312,A -85,B 0,C 180,E1 -19850.137,E2 -19850.137} C_VEL
LIN {X 0,Y 252.691,Z 615.035,A -85,B 0,C 180,E1 -19852.275,E2 -19852.275} C_VEL
LIN {X 0,Y 247.527,Z 627.666,A -85,B 0,C 180,E1 -19854.904,E2 -19854.904} C_VEL
LIN {X 0,Y 242.992,Z 638.442,A -85,B 0,C 180,E1 -19857.652,E2 -19857.652} C_VEL
LIN {X 0,Y 238.259,Z 648.843,A -85,B 0,C 180,E1 -19860.876,E2 -19860.876} C_VEL
LIN {X 0,Y 234.285,Z 657.699,A -85,B 0,C 180,E1 -19864.296,E2 -19864.296} C_VEL
LIN {X 0,Y 231.272,Z 664.813,A -85,B 0,C 180,E1 -19867.676,E2 -19867.676} C_VEL
LIN {X 0,Y 228.881,Z 670.863,A -85,B 0,C 180,E1 -19871.191,E2 -19871.191} C_VEL
LIN {X 0,Y 226.93,Z 676.736,A -85,B 0,C 180,E1 -19875.655,E2 -19875.655} C_VEL
LIN {X 0,Y 225.963,Z 680.173,A -85,B 0,C 180,E1 -19879.245,E2 -19879.245} C_VEL
LIN {X 0,Y 225.587,Z 682.68,A -85,B 0,C 180,E1 -19882.841,E2 -19882.841} C_VEL
LIN {X 0,Y 225.581,Z 684.099,A -85,B 0,C 180,E1 -19886.428,E2 -19886.428} C_VEL
LIN {X 0,Y 225.713,Z 684.633,A -85,B 0,C 180,E1 -19890,E2 -19890} C_VEL
LIN {X 0,Y 225.581,Z 684.088,A -85,B 0,C 180,E1 -19893.572,E2 -19893.572} C_VEL
LIN {X 0,Y 225.587,Z 682.657,A -85,B 0,C 180,E1 -19897.159,E2 -19897.159} C_VEL
LIN {X 0,Y 225.963,Z 680.141,A -85,B 0,C 180,E1 -19900.755,E2 -19900.755} C_VEL
LIN {X 0,Y 227.238,Z 675.609,A -85,B 0,C 180,E1 -19905.241,E2 -19905.241} C_VEL
LIN {X 0,Y 228.88,Z 670.805,A -85,B 0,C 180,E1 -19908.809,E2 -19908.809} C_VEL
LIN {X 0,Y 232.012,Z 663.083,A -85,B 0,C 180,E1 -19913.19,E2 -19913.19} C_VEL
LIN {X 0,Y 235.775,Z 654.384,A -85,B 0,C 180,E1 -19917.037,E2 -19917.037} C_VEL
LIN {X 0,Y 239.942,Z 645.004,A -85,B 0,C 180,E1 -19920.348,E2 -19920.348} C_VEL
LIN {X 0,Y 244.129,Z 635.357,A -85,B 0,C 180,E1 -19923.159,E2 -19923.159} C_VEL
LIN {X 0,Y 248.936,Z 624.126,A -85,B 0,C 180,E1 -19925.86,E2 -19925.86} C_VEL
LIN {X 0,Y 253.864,Z 611.899,A -85,B 0,C 180,E1 -19928.274,E2 -19928.274} C_VEL
LIN {X 0,Y 258.445,Z 599.811,A -85,B 0,C 180,E1 -19930.209,E2 -19930.209} C_VEL
LIN {X 0,Y 262.914,Z 586.872,A -85,B 0,C 180,E1 -19931.934,E2 -19931.934} C_VEL
LIN {X 0,Y 267.086,Z 573.243,A -85,B 0,C 180,E1 -19933.428,E2 -19933.428} C_VEL
LIN {X 0,Y 270.96,Z 558.544,A -85,B 0,C 180,E1 -19934.712,E2 -19934.712} C_VEL
LIN {X 0,Y 274.406,Z 542.596,A -85,B 0,C 180,E1 -19935.817,E2 -19935.817} C_VEL
LIN {X 0,Y 277.386,Z 525.763,A -85,B 0,C 180,E1 -19936.656,E2 -19936.656} C_VEL
LIN {X 0,Y 279.435,Z 509.095,A -85,B 0,C 180,E1 -19937.243,E2 -19937.243} C_VEL
LIN {X 0,Y 286.581,Z 393.492,A -85,B 0,C 180,E1 -19939.998,E2 -19939.998} C_VEL
LIN {X 0,Y 281.981,Z 383.439,A -85,B 0,C 180,E1 -19941.515,E2 -19941.515} C_VEL
LIN {X 0,Y 276.454,Z 372.588,A -85,B 0,C 180,E1 -19943.426,E2 -19943.426} C_VEL
LIN {X 0,Y 270.91,Z 362.474,A -85,B 0,C 180,E1 -19945.482,E2 -19945.482} C_VEL
LIN {X 0,Y 266.516,Z 355.154,A -85,B 0,C 180,E1 -19947.221,E2 -19947.221} C_VEL
LIN {X 0,Y 261.631,Z 347.37,A -85,B 0,C 180,E1 -19949.311,E2 -19949.311} C_VEL
LIN {X 0,Y 257.927,Z 342.467,A -85,B 0,C 180,E1 -19950.986,E2 -19950.986} C_VEL
LIN {X 0,Y 254.844,Z 338.415,A -85,B 0,C 180,E1 -19952.489,E2 -19952.489} C_VEL
LIN {X 0,Y 251.459,Z 334.023,A -85,B 0,C 180,E1 -19954.273,E2 -19954.273} C_VEL
LIN {X 0,Y 248.463,Z 330.381,A -85,B 0,C 180,E1 -19955.981,E2 -19955.981} C_VEL
LIN {X 0,Y 247.659,Z 329.189,A -85,B 0,C 180,E1 -19956.481,E2 -19956.481} C_VEL
LIN {X 0,Y 244.82,Z 326.371,A -85,B 0,C 180,E1 -19958.255,E2 -19958.255} C_VEL
LIN {X 0,Y 243.372,Z 323.926,A -85,B 0,C 180,E1 -19959.312,E2 -19959.312} C_VEL
LIN {X 0,Y 240.671,Z 321.715,A -85,B 0,C 180,E1 -19961.264,E2 -19961.264} C_VEL
LIN {X 0,Y 238.905,Z 318.653,A -85,B 0,C 180,E1 -19962.837,E2 -19962.837} C_VEL
LIN {X 0,Y 235.272,Z 315.756,A -85,B 0,C 180,E1 -19966.284,E2 -19966.284} C_VEL
LIN {X 0,Y 233.921,Z 312.961,A -85,B 0,C 180,E1 -19968.08,E2 -19968.08} C_VEL
LIN {X 0,Y 233.794,Z 312.489,A -85,B 0,C 180,E1 -19968.293,E2 -19968.293} C_VEL
LIN {X 0,Y 229.368,Z 309.047,A -85,B 0,C 180,E1 -19977.805,E2 -19977.805} C_VEL
LIN {X 0,Y 229.244,Z 308.403,A -85,B 0,C 180,E1 -19980,E2 -19980} C_VEL
LIN {X 0,Y 229.333,Z 309.028,A -85,B 0,C 180,E1 -19982.415,E2 -19982.415} C_VEL
LIN {X 0,Y 233.813,Z 312.612,A -85,B 0,C 180,E1 -19992.202,E2 -19992.202} C_VEL
LIN {X 0,Y 234.993,Z 315.348,A -85,B 0,C 180,E1 -19993.843,E2 -19993.843} C_VEL
LIN {X 0,Y 237.356,Z 317.638,A -85,B 0,C 180,E1 -19996.274,E2 -19996.274} C_VEL
LIN {X 0,Y 238.891,Z 318.628,A -85,B 0,C 180,E1 -19997.606,E2 -19997.606} C_VEL
LIN {X 0,Y 240.653,Z 321.722,A -85,B 0,C 180,E1 -19999.181,E2 -19999.181} C_VEL
LIN {X 0,Y 243.65,Z 324.387,A -85,B 0,C 180,E1 -20001.35,E2 -20001.35} C_VEL
LIN {X 0,Y 245.983,Z 327.751,A -85,B 0,C 180,E1 -20002.966,E2 -20002.966} C_VEL
LIN {X 0,Y 248.189,Z 329.86,A -85,B 0,C 180,E1 -20004.298,E2 -20004.298} C_VEL
LIN {X 0,Y 250.875,Z 333.449,A -85,B 0,C 180,E1 -20005.87,E2 -20005.87} C_VEL
LIN {X 0,Y 252.295,Z 335.06,A -85,B 0,C 180,E1 -20006.636,E2 -20006.636} C_VEL
LIN {X 0,Y 255.376,Z 338.979,A -85,B 0,C 180,E1 -20008.226,E2 -20008.226} C_VEL
LIN {X 0,Y 260.347,Z 345.651,A -85,B 0,C 180,E1 -20010.578,E2 -20010.578} C_VEL
LIN {X 0,Y 265.247,Z 352.316,A -85,B 0,C 180,E1 -20012.671,E2 -20012.671} C_VEL
LIN {X 0,Y 273.034,Z 363.908,A -85,B 0,C 180,E1 -20015.675,E2 -20015.675} C_VEL
LIN {X 0,Y 281.197,Z 377.409,A -85,B 0,C 180,E1 -20018.498,E2 -20018.498} C_VEL
LIN {X 0,Y 286.827,Z 387.471,A -85,B 0,C 180,E1 -20020.287,E2 -20020.287} C_VEL
LIN {X 0,Y 280.004,Z 497.934,A -85,B 0,C 180,E1 -20022.925,E2 -20022.925} C_VEL
LIN {X 0,Y 278.087,Z 514.458,A -85,B 0,C 180,E1 -20023.531,E2 -20023.531} C_VEL
LIN {X 0,Y 275.405,Z 530.94,A -85,B 0,C 180,E1 -20024.396,E2 -20024.396} C_VEL
LIN {X 0,Y 272.112,Z 546.909,A -85,B 0,C 180,E1 -20025.527,E2 -20025.527} C_VEL
LIN {X 0,Y 268.815,Z 559.878,A -85,B 0,C 180,E1 -20026.663,E2 -20026.663} C_VEL
LIN {X 0,Y 264.773,Z 573.777,A -85,B 0,C 180,E1 -20028.181,E2 -20028.181} C_VEL
LIN {X 0,Y 260.115,Z 587.926,A -85,B 0,C 180,E1 -20030.082,E2 -20030.082} C_VEL
LIN {X 0,Y 256.07,Z 598.974,A -85,B 0,C 180,E1 -20031.865,E2 -20031.865} C_VEL
LIN {X 0,Y 251.044,Z 611.372,A -85,B 0,C 180,E1 -20034.278,E2 -20034.278} C_VEL
LIN {X 0,Y 246.045,Z 623.22,A -85,B 0,C 180,E1 -20037.132,E2 -20037.132} C_VEL
LIN {X 0,Y 241.111,Z 633.96,A -85,B 0,C 180,E1 -20040.296,E2 -20040.296} C_VEL
LIN {X 0,Y 237.045,Z 642.968,A -85,B 0,C 180,E1 -20043.594,E2 -20043.594} C_VEL
LIN {X 0,Y 233.557,Z 650.494,A -85,B 0,C 180,E1 -20046.972,E2 -20046.972} C_VEL
LIN {X 0,Y 230.375,Z 657.616,A -85,B 0,C 180,E1 -20051.034,E2 -20051.034} C_VEL
LIN {X 0,Y 228.265,Z 662.723,A -85,B 0,C 180,E1 -20054.829,E2 -20054.829} C_VEL
LIN {X 0,Y 226.698,Z 667.12,A -85,B 0,C 180,E1 -20059.28,E2 -20059.28} C_VEL
LIN {X 0,Y 226.011,Z 669.55,A -85,B 0,C 180,E1 -20062.855,E2 -20062.855} C_VEL
LIN {X 0,Y 225.733,Z 670.924,A -85,B 0,C 180,E1 -20066.43,E2 -20066.43} C_VEL
LIN {X 0,Y 225.744,Z 671.451,A -85,B 0,C 180,E1 -20070,E2 -20070} C_VEL
LIN {X 0,Y 225.733,Z 670.96,A -85,B 0,C 180,E1 -20073.57,E2 -20073.57} C_VEL
LIN {X 0,Y 226.01,Z 669.619,A -85,B 0,C 180,E1 -20077.145,E2 -20077.145} C_VEL
LIN {X 0,Y 226.687,Z 667.224,A -85,B 0,C 180,E1 -20080.72,E2 -20080.72} C_VEL
LIN {X 0,Y 227.789,Z 663.922,A -85,B 0,C 180,E1 -20084.29,E2 -20084.29} C_VEL
LIN {X 0,Y 229.612,Z 659.464,A -85,B 0,C 180,E1 -20087.823,E2 -20087.823} C_VEL
LIN {X 0,Y 232.034,Z 653.943,A -85,B 0,C 180,E1 -20091.313,E2 -20091.313} C_VEL
LIN {X 0,Y 235.133,Z 647.174,A -85,B 0,C 180,E1 -20094.737,E2 -20094.737} C_VEL
LIN {X 0,Y 238.907,Z 638.976,A -85,B 0,C 180,E1 -20098.078,E2 -20098.078} C_VEL
LIN {X 0,Y 243.396,Z 629.208,A -85,B 0,C 180,E1 -20101.315,E2 -20101.315} C_VEL
LIN {X 0,Y 247.902,Z 619.157,A -85,B 0,C 180,E1 -20104.049,E2 -20104.049} C_VEL
LIN {X 0,Y 252.863,Z 607.308,A -85,B 0,C 180,E1 -20106.695,E2 -20106.695} C_VEL
LIN {X 0,Y 257.898,Z 594.258,A -85,B 0,C 180,E1 -20109.063,E2 -20109.063} C_VEL
LIN {X 0,Y 262.555,Z 581.213,A -85,B 0,C 180,E1 -20110.98,E2 -20110.98} C_VEL
LIN {X 0,Y 266.468,Z 568.534,A -85,B 0,C 180,E1 -20112.559,E2 -20112.559} C_VEL
LIN {X 0,Y 270.531,Z 553.823,A -85,B 0,C 180,E1 -20114.021,E2 -20114.021} C_VEL
LIN {X 0,Y 274.117,Z 538.404,A -85,B 0,C 180,E1 -20115.224,E2 -20115.224} C_VEL
LIN {X 0,Y 276.937,Z 522.727,A -85,B 0,C 180,E1 -20116.192,E2 -20116.192} C_VEL
LIN {X 0,Y 279.204,Z 507.06,A -85,B 0,C 180,E1 -20116.884,E2 -20116.884} C_VEL
LIN {X 0,Y 280.703,Z 490.477,A -85,B 0,C 180,E1 -20117.393,E2 -20117.393} C_VEL
LIN {X 0,Y 286.959,Z 387.626,A -85,B 0,C 180,E1 -20119.824,E2 -20119.824} C_VEL
LIN {X 0,Y 280.115,Z 375.483,A -85,B 0,C 180,E1 -20122.017,E2 -20122.017} C_VEL
LIN {X 0,Y 272.438,Z 362.991,A -85,B 0,C 180,E1 -20124.708,E2 -20124.708} C_VEL
LIN {X 0,Y 266.399,Z 354.009,A -85,B 0,C 180,E1 -20127.035,E2 -20127.035} C_VEL
LIN {X 0,Y 261.589,Z 347.281,A -85,B 0,C 180,E1 -20129.061,E2 -20129.061} C_VEL
LIN {X 0,Y 258,Z 342.483,A -85,B 0,C 180,E1 -20130.696,E2 -20130.696} C_VEL
LIN {X 0,Y 254.984,Z 338.536,A -85,B 0,C 180,E1 -20132.17,E2 -20132.17} C_VEL
LIN {X 0,Y 252.034,Z 334.538,A -85,B 0,C 180,E1 -20133.732,E2 -20133.732} C_VEL
LIN {X 0,Y 248.813,Z 330.82,A -85,B 0,C 180,E1 -20135.545,E2 -20135.545} C_VEL
LIN {X 0,Y 247.661,Z 329.185,A -85,B 0,C 180,E1 -20136.259,E2 -20136.259} C_VEL
LIN {X 0,Y 244.779,Z 326.252,A -85,B 0,C 180,E1 -20138.084,E2 -20138.084} C_VEL
LIN {X 0,Y 243.301,Z 323.875,A -85,B 0,C 180,E1 -20139.168,E2 -20139.168} C_VEL
LIN {X 0,Y 240.73,Z 321.789,A -85,B 0,C 180,E1 -20141.047,E2 -20141.047} C_VEL
LIN {X 0,Y 238.981,Z 318.762,A -85,B 0,C 180,E1 -20142.622,E2 -20142.622} C_VEL
LIN {X 0,Y 238.344,Z 318.147,A -85,B 0,C 180,E1 -20143.187,E2 -20143.187} C_VEL
LIN {X 0,Y 235.574,Z 316.141,A -85,B 0,C 180,E1 -20145.862,E2 -20145.862} C_VEL
LIN {X 0,Y 235.399,Z 315.931,A -85,B 0,C 180,E1 -20146.06,E2 -20146.06} C_VEL
LIN {X 0,Y 234.128,Z 315.407,A -85,B 0,C 180,E1 -20147.467,E2 -20147.467} C_VEL
LIN {X 0,Y 232.098,Z 316.357,A -85,B 0,C 180,E1 -20149.848,E2 -20149.848} C_VEL
LIN {X 0,Y 230.152,Z 317.836,A -85,B 0,C 180,E1 -20152.768,E2 -20152.768} C_VEL
LIN {X 0,Y 229.7,Z 317.799,A -85,B 0,C 180,E1 -20153.758,E2 -20153.758} C_VEL
LIN {X 0,Y 228.641,Z 316.108,A -85,B 0,C 180,E1 -20159.119,E2 -20159.119} C_VEL
LIN {X 0,Y 228.747,Z 316.435,A -85,B 0,C 180,E1 -20161.981,E2 -20161.981} C_VEL
LIN {X 0,Y 232.649,Z 319.612,A -85,B 0,C 180,E1 -20171.048,E2 -20171.048} C_VEL
LIN {X 0,Y 233.932,Z 322.42,A -85,B 0,C 180,E1 -20172.911,E2 -20172.911} C_VEL
LIN {X 0,Y 236.667,Z 324.881,A -85,B 0,C 180,E1 -20175.774,E2 -20175.774} C_VEL
LIN {X 0,Y 237.507,Z 325.536,A -85,B 0,C 180,E1 -20176.537,E2 -20176.537} C_VEL
LIN {X 0,Y 239.409,Z 328.681,A -85,B 0,C 180,E1 -20178.284,E2 -20178.284} C_VEL
LIN {X 0,Y 242.051,Z 331.15,A -85,B 0,C 180,E1 -20180.28,E2 -20180.28} C_VEL
LIN {X 0,Y 244.533,Z 334.609,A -85,B 0,C 180,E1 -20182.05,E2 -20182.05} C_VEL
LIN {X 0,Y 246.37,Z 336.431,A -85,B 0,C 180,E1 -20183.204,E2 -20183.204} C_VEL
LIN {X 0,Y 249.032,Z 339.992,A -85,B 0,C 180,E1 -20184.821,E2 -20184.821} C_VEL
LIN {X 0,Y 250.653,Z 342.001,A -85,B 0,C 180,E1 -20185.733,E2 -20185.733} C_VEL
LIN {X 0,Y 254.337,Z 346.875,A -85,B 0,C 180,E1 -20187.682,E2 -20187.682} C_VEL
LIN {X 0,Y 257.929,Z 351.764,A -85,B 0,C 180,E1 -20189.427,E2 -20189.427} C_VEL
LIN {X 0,Y 260.899,Z 356.131,A -85,B 0,C 180,E1 -20190.784,E2 -20190.784} C_VEL
LIN {X 0,Y 266.513,Z 365.552,A -85,B 0,C 180,E1 -20193.195,E2 -20193.195} C_VEL
LIN {X 0,Y 272.425,Z 376.333,A -85,B 0,C 180,E1 -20195.518,E2 -20195.518} C_VEL
LIN {X 0,Y 278.771,Z 388.979,A -85,B 0,C 180,E1 -20197.816,E2 -20197.816} C_VEL
LIN {X 0,Y 282.032,Z 396.29,A -85,B 0,C 180,E1 -20198.946,E2 -20198.946} C_VEL
LIN {X 0,Y 274.779,Z 508.976,A -85,B 0,C 180,E1 -20201.642,E2 -20201.642} C_VEL
LIN {X 0,Y 272.745,Z 525.277,A -85,B 0,C 180,E1 -20202.223,E2 -20202.223} C_VEL
LIN {X 0,Y 269.763,Z 541.744,A -85,B 0,C 180,E1 -20203.034,E2 -20203.034} C_VEL
LIN {X 0,Y 266.401,Z 556.761,A -85,B 0,C 180,E1 -20204.038,E2 -20204.038} C_VEL
LIN {X 0,Y 262.445,Z 571.713,A -85,B 0,C 180,E1 -20205.337,E2 -20205.337} C_VEL
LIN {X 0,Y 257.616,Z 586.954,A -85,B 0,C 180,E1 -20206.999,E2 -20206.999} C_VEL
LIN {X 0,Y 252.758,Z 600.653,A -85,B 0,C 180,E1 -20208.875,E2 -20208.875} C_VEL
LIN {X 0,Y 247.888,Z 612.868,A -85,B 0,C 180,E1 -20210.89,E2 -20210.89} C_VEL
LIN {X 0,Y 243.183,Z 624.095,A -85,B 0,C 180,E1 -20213.154,E2 -20213.154} C_VEL
LIN {X 0,Y 238.223,Z 635.294,A -85,B 0,C 180,E1 -20215.908,E2 -20215.908} C_VEL
LIN {X 0,Y 233.119,Z 646.151,A -85,B 0,C 180,E1 -20219.169,E2 -20219.169} C_VEL
LIN {X 0,Y 228.865,Z 655.288,A -85,B 0,C 180,E1 -20222.573,E2 -20222.573} C_VEL
LIN {X 0,Y 225.371,Z 662.954,A -85,B 0,C 180,E1 -20226.085,E2 -20226.085} C_VEL
LIN {X 0,Y 222.074,Z 670.654,A -85,B 0,C 180,E1 -20230.592,E2 -20230.592} C_VEL
LIN {X 0,Y 219.96,Z 676.526,A -85,B 0,C 180,E1 -20235.19,E2 -20235.19} C_VEL
LIN {X 0,Y 218.927,Z 679.965,A -85,B 0,C 180,E1 -20238.895,E2 -20238.895} C_VEL
LIN {X 0,Y 218.522,Z 682.472,A -85,B 0,C 180,E1 -20242.609,E2 -20242.609} C_VEL
LIN {X 0,Y 218.496,Z 683.892,A -85,B 0,C 180,E1 -20246.312,E2 -20246.312} C_VEL
LIN {X 0,Y 218.628,Z 684.427,A -85,B 0,C 180,E1 -20250,E2 -20250} C_VEL
LIN {X 0,Y 218.481,Z 683.717,A -85,B 0,C 180,E1 -20254.301,E2 -20254.301} C_VEL
LIN {X 0,Y 218.522,Z 682.449,A -85,B 0,C 180,E1 -20257.391,E2 -20257.391} C_VEL
LIN {X 0,Y 218.927,Z 679.931,A -85,B 0,C 180,E1 -20261.105,E2 -20261.105} C_VEL
LIN {X 0,Y 219.955,Z 676.481,A -85,B 0,C 180,E1 -20264.81,E2 -20264.81} C_VEL
LIN {X 0,Y 222.074,Z 670.594,A -85,B 0,C 180,E1 -20269.408,E2 -20269.408} C_VEL
LIN {X 0,Y 225.388,Z 662.871,A -85,B 0,C 180,E1 -20273.914,E2 -20273.914} C_VEL
LIN {X 0,Y 229.371,Z 654.172,A -85,B 0,C 180,E1 -20277.857,E2 -20277.857} C_VEL
LIN {X 0,Y 233.747,Z 644.791,A -85,B 0,C 180,E1 -20281.241,E2 -20281.241} C_VEL
LIN {X 0,Y 238.107,Z 635.143,A -85,B 0,C 180,E1 -20284.111,E2 -20284.111} C_VEL
LIN {X 0,Y 243.144,Z 623.914,A -85,B 0,C 180,E1 -20286.853,E2 -20286.853} C_VEL
LIN {X 0,Y 248.265,Z 611.687,A -85,B 0,C 180,E1 -20289.301,E2 -20289.301} C_VEL
LIN {X 0,Y 253.194,Z 599.06,A -85,B 0,C 180,E1 -20291.342,E2 -20291.342} C_VEL
LIN {X 0,Y 258.114,Z 585.227,A -85,B 0,C 180,E1 -20293.165,E2 -20293.165} C_VEL
LIN {X 0,Y 262.429,Z 571.338,A -85,B 0,C 180,E1 -20294.667,E2 -20294.667} C_VEL
LIN {X 0,Y 266.706,Z 555.332,A -85,B 0,C 180,E1 -20296.031,E2 -20296.031} C_VEL
LIN {X 0,Y 270,Z 540.027,A -85,B 0,C 180,E1 -20297.035,E2 -20297.035} C_VEL
LIN {X 0,Y 272.809,Z 523.806,A -85,B 0,C 180,E1 -20297.814,E2 -20297.814} C_VEL
LIN {X 0,Y 274.767,Z 507.379,A -85,B 0,C 180,E1 -20298.375,E2 -20298.375} C_VEL
LIN {X 0,Y 281.896,Z 396.161,A -85,B 0,C 180,E1 -20301.032,E2 -20301.032} C_VEL
LIN {X 0,Y 276.673,Z 384.834,A -85,B 0,C 180,E1 -20302.85,E2 -20302.85} C_VEL
LIN {X 0,Y 269.861,Z 371.612,A -85,B 0,C 180,E1 -20305.385,E2 -20305.385} C_VEL
LIN {X 0,Y 264.177,Z 361.671,A -85,B 0,C 180,E1 -20307.686,E2 -20307.686} C_VEL
LIN {X 0,Y 258.999,Z 353.236,A -85,B 0,C 180,E1 -20309.98,E2 -20309.98} C_VEL
LIN {X 0,Y 255.508,Z 348.542,A -85,B 0,C 180,E1 -20311.619,E2 -20311.619} C_VEL
LIN {X 0,Y 252.381,Z 344.323,A -85,B 0,C 180,E1 -20313.207,E2 -20313.207} C_VEL
LIN {X 0,Y 249.493,Z 340.478,A -85,B 0,C 180,E1 -20314.789,E2 -20314.789} C_VEL
LIN {X 0,Y 246.387,Z 336.563,A -85,B 0,C 180,E1 -20316.63,E2 -20316.63} C_VEL
LIN {X 0,Y 245.237,Z 335.238,A -85,B 0,C 180,E1 -20317.351,E2 -20317.351} C_VEL
LIN {X 0,Y 242.588,Z 332.145,A -85,B 0,C 180,E1 -20319.13,E2 -20319.13} C_VEL
LIN {X 0,Y 241.713,Z 330.619,A -85,B 0,C 180,E1 -20319.802,E2 -20319.802} C_VEL
LIN {X 0,Y 238.943,Z 328.107,A -85,B 0,C 180,E1 -20321.901,E2 -20321.901} C_VEL
LIN {X 0,Y 237.288,Z 325.162,A -85,B 0,C 180,E1 -20323.448,E2 -20323.448} C_VEL
LIN {X 0,Y 234.403,Z 323.043,A -85,B 0,C 180,E1 -20326.233,E2 -20326.233} C_VEL
LIN {X 0,Y 232.682,Z 319.869,A -85,B 0,C 180,E1 -20328.512,E2 -20328.512} C_VEL
LIN {X 0,Y 232.266,Z 319.346,A -85,B 0,C 180,E1 -20329.099,E2 -20329.099} C_VEL
LIN {X 0,Y 228.378,Z 315.459,A -85,B 0,C 180,E1 -20340,E2 -20340} C_VEL
LIN {X 0,Y 228.485,Z 316.226,A -85,B 0,C 180,E1 -20342.645,E2 -20342.645} C_VEL
LIN {X 0,Y 232.645,Z 319.712,A -85,B 0,C 180,E1 -20351.877,E2 -20351.877} C_VEL
LIN {X 0,Y 233.945,Z 322.415,A -85,B 0,C 180,E1 -20353.685,E2 -20353.685} C_VEL
LIN {X 0,Y 236.236,Z 324.601,A -85,B 0,C 180,E1 -20356.079,E2 -20356.079} C_VEL
LIN {X 0,Y 237.413,Z 325.429,A -85,B 0,C 180,E1 -20357.135,E2 -20357.135} C_VEL
LIN {X 0,Y 239.541,Z 328.857,A -85,B 0,C 180,E1 -20359.051,E2 -20359.051} C_VEL
LIN {X 0,Y 241.924,Z 330.97,A -85,B 0,C 180,E1 -20360.817,E2 -20360.817} C_VEL
LIN {X 0,Y 244.456,Z 334.54,A -85,B 0,C 180,E1 -20362.614,E2 -20362.614} C_VEL
LIN {X 0,Y 246.305,Z 336.378,A -85,B 0,C 180,E1 -20363.768,E2 -20363.768} C_VEL
LIN {X 0,Y 249.22,Z 340.191,A -85,B 0,C 180,E1 -20365.515,E2 -20365.515} C_VEL
LIN {X 0,Y 250.65,Z 342.128,A -85,B 0,C 180,E1 -20366.322,E2 -20366.322} C_VEL
LIN {X 0,Y 254.139,Z 346.664,A -85,B 0,C 180,E1 -20368.155,E2 -20368.155} C_VEL
LIN {X 0,Y 257.959,Z 351.825,A -85,B 0,C 180,E1 -20370,E2 -20370} C_VEL
LIN {X 0,Y 262.94,Z 358.833,A -85,B 0,C 180,E1 -20372.202,E2 -20372.202} C_VEL
LIN {X 0,Y 270.051,Z 369.627,A -85,B 0,C 180,E1 -20375.038,E2 -20375.038} C_VEL
LIN {X 0,Y 278.189,Z 383.363,A -85,B 0,C 180,E1 -20377.952,E2 -20377.952} C_VEL
LIN {X 0,Y 282.073,Z 390.439,A -85,B 0,C 180,E1 -20379.242,E2 -20379.242} C_VEL
LIN {X 0,Y 275.253,Z 497.81,A -85,B 0,C 180,E1 -20381.835,E2 -20381.835} C_VEL
LIN {X 0,Y 273.396,Z 513.762,A -85,B 0,C 180,E1 -20382.418,E2 -20382.418} C_VEL
LIN {X 0,Y 270.737,Z 529.86,A -85,B 0,C 180,E1 -20383.242,E2 -20383.242} C_VEL
LIN {X 0,Y 267.593,Z 545.144,A -85,B 0,C 180,E1 -20384.301,E2 -20384.301} C_VEL
LIN {X 0,Y 263.703,Z 560.091,A -85,B 0,C 180,E1 -20385.606,E2 -20385.606} C_VEL
LIN {X 0,Y 259.534,Z 573.916,A -85,B 0,C 180,E1 -20387.124,E2 -20387.124} C_VEL
LIN {X 0,Y 254.706,Z 588.137,A -85,B 0,C 180,E1 -20389.056,E2 -20389.056} C_VEL
LIN {X 0,Y 250.494,Z 599.186,A -85,B 0,C 180,E1 -20390.856,E2 -20390.856} C_VEL
LIN {X 0,Y 245.737,Z 610.56,A -85,B 0,C 180,E1 -20393.088,E2 -20393.088} C_VEL
LIN {X 0,Y 240.718,Z 621.958,A -85,B 0,C 180,E1 -20395.805,E2 -20395.805} C_VEL
LIN {X 0,Y 236.157,Z 631.719,A -85,B 0,C 180,E1 -20398.614,E2 -20398.614} C_VEL
LIN {X 0,Y 231.581,Z 641.254,A -85,B 0,C 180,E1 -20402.017,E2 -20402.017} C_VEL
LIN {X 0,Y 227.801,Z 648.917,A -85,B 0,C 180,E1 -20405.387,E2 -20405.387} C_VEL
LIN {X 0,Y 224.706,Z 655.447,A -85,B 0,C 180,E1 -20408.92,E2 -20408.92} C_VEL
LIN {X 0,Y 222.309,Z 660.724,A -85,B 0,C 180,E1 -20412.523,E2 -20412.523} C_VEL
LIN {X 0,Y 220.912,Z 663.984,A -85,B 0,C 180,E1 -20415.256,E2 -20415.256} C_VEL
LIN {X 0,Y 219.678,Z 667.329,A -85,B 0,C 180,E1 -20418.933,E2 -20418.933} C_VEL
LIN {X 0,Y 218.949,Z 669.758,A -85,B 0,C 180,E1 -20422.623,E2 -20422.623} C_VEL
LIN {X 0,Y 218.647,Z 671.132,A -85,B 0,C 180,E1 -20426.314,E2 -20426.314} C_VEL
LIN {X 0,Y 218.659,Z 671.658,A -85,B 0,C 180,E1 -20430,E2 -20430} C_VEL
LIN {X 0,Y 218.647,Z 671.167,A -85,B 0,C 180,E1 -20433.686,E2 -20433.686} C_VEL
LIN {X 0,Y 218.948,Z 669.827,A -85,B 0,C 180,E1 -20437.377,E2 -20437.377} C_VEL
LIN {X 0,Y 219.667,Z 667.433,A -85,B 0,C 180,E1 -20441.067,E2 -20441.067} C_VEL
LIN {X 0,Y 220.88,Z 664.129,A -85,B 0,C 180,E1 -20444.746,E2 -20444.746} C_VEL
LIN {X 0,Y 223.424,Z 658.396,A -85,B 0,C 180,E1 -20449.321,E2 -20449.321} C_VEL
LIN {X 0,Y 226.902,Z 650.956,A -85,B 0,C 180,E1 -20453.744,E2 -20453.744} C_VEL
LIN {X 0,Y 230.595,Z 643.46,A -85,B 0,C 180,E1 -20457.204,E2 -20457.204} C_VEL
LIN {X 0,Y 234.841,Z 634.514,A -85,B 0,C 180,E1 -20460.58,E2 -20460.58} C_VEL
LIN {X 0,Y 239.93,Z 623.845,A -85,B 0,C 180,E1 -20463.817,E2 -20463.817} C_VEL
LIN {X 0,Y 244.796,Z 613.05,A -85,B 0,C 180,E1 -20466.499,E2 -20466.499} C_VEL
LIN {X 0,Y 250.364,Z 599.776,A -85,B 0,C 180,E1 -20469.168,E2 -20469.168} C_VEL
LIN {X 0,Y 255.479,Z 586.446,A -85,B 0,C 180,E1 -20471.316,E2 -20471.316} C_VEL
LIN {X 0,Y 259.826,Z 573.248,A -85,B 0,C 180,E1 -20473.087,E2 -20473.087} C_VEL
LIN {X 0,Y 264.518,Z 557.544,A -85,B 0,C 180,E1 -20474.755,E2 -20474.755} C_VEL
LIN {X 0,Y 268.212,Z 543.106,A -85,B 0,C 180,E1 -20475.967,E2 -20475.967} C_VEL
LIN {X 0,Y 271.337,Z 527.38,A -85,B 0,C 180,E1 -20477.03,E2 -20477.03} C_VEL
LIN {X 0,Y 273.901,Z 511.172,A -85,B 0,C 180,E1 -20477.808,E2 -20477.808} C_VEL
LIN {X 0,Y 275.603,Z 494.902,A -85,B 0,C 180,E1 -20478.365,E2 -20478.365} C_VEL
LIN {X 0,Y 282.22,Z 390.596,A -85,B 0,C 180,E1 -20480.867,E2 -20480.867} C_VEL
LIN {X 0,Y 275.556,Z 378.714,A -85,B 0,C 180,E1 -20483.119,E2 -20483.119} C_VEL
LIN {X 0,Y 269.095,Z 368.102,A -85,B 0,C 180,E1 -20485.495,E2 -20485.495} C_VEL
LIN {X 0,Y 262.357,Z 357.845,A -85,B 0,C 180,E1 -20488.235,E2 -20488.235} C_VEL
LIN {X 0,Y 256.321,Z 349.424,A -85,B 0,C 180,E1 -20490.979,E2 -20490.979} C_VEL
LIN {X 0,Y 252.418,Z 344.351,A -85,B 0,C 180,E1 -20492.943,E2 -20492.943} C_VEL
LIN {X 0,Y 249.349,Z 340.289,A -85,B 0,C 180,E1 -20494.638,E2 -20494.638} C_VEL
LIN {X 0,Y 246.329,Z 336.359,A -85,B 0,C 180,E1 -20496.457,E2 -20496.457} C_VEL
LIN {X 0,Y 242.727,Z 332.282,A -85,B 0,C 180,E1 -20498.839,E2 -20498.839} C_VEL
LIN {X 0,Y 241.759,Z 330.648,A -85,B 0,C 180,E1 -20499.583,E2 -20499.583} C_VEL
LIN {X 0,Y 239.132,Z 328.333,A -85,B 0,C 180,E1 -20501.582,E2 -20501.582} C_VEL
LIN {X 0,Y 237.151,Z 325.055,A -85,B 0,C 180,E1 -20503.437,E2 -20503.437} C_VEL
LIN {X 0,Y 234.345,Z 322.945,A -85,B 0,C 180,E1 -20506.229,E2 -20506.229} C_VEL
LIN {X 0,Y 232.85,Z 320.241,A -85,B 0,C 180,E1 -20508.245,E2 -20508.245} C_VEL
LIN {X 0,Y 232.596,Z 319.477,A -85,B 0,C 180,E1 -20508.673,E2 -20508.673} C_VEL
LIN {X 0,Y 229.7,Z 317.799,A -85,B 0,C 180,E1 -20513.758,E2 -20513.758} C_VEL
LIN {X 0,Y 229.129,Z 317.983,A -85,B 0,C 180,E1 -20515.228,E2 -20515.228} C_VEL
LIN {X 0,Y 228.312,Z 319.98,A -85,B 0,C 180,E1 -20517.651,E2 -20517.651} C_VEL
LIN {X 0,Y 227.819,Z 322.832,A -85,B 0,C 180,E1 -20520.577,E2 -20520.577} C_VEL
LIN {X 0,Y 227.841,Z 323.361,A -85,B 0,C 180,E1 -20521.572,E2 -20521.572} C_VEL
LIN {X 0,Y 231.442,Z 326.494,A -85,B 0,C 180,E1 -20530.608,E2 -20530.608} C_VEL
LIN {X 0,Y 233.059,Z 329.71,A -85,B 0,C 180,E1 -20532.96,E2 -20532.96} C_VEL
LIN {X 0,Y 236.084,Z 332.376,A -85,B 0,C 180,E1 -20536.089,E2 -20536.089} C_VEL
LIN {X 0,Y 238.182,Z 335.643,A -85,B 0,C 180,E1 -20538.048,E2 -20538.048} C_VEL
LIN {X 0,Y 240.38,Z 337.741,A -85,B 0,C 180,E1 -20539.758,E2 -20539.758} C_VEL
LIN {X 0,Y 243.089,Z 341.47,A -85,B 0,C 180,E1 -20541.74,E2 -20541.74} C_VEL
LIN {X 0,Y 244.585,Z 343.059,A -85,B 0,C 180,E1 -20542.713,E2 -20542.713} C_VEL
LIN {X 0,Y 247.691,Z 347.038,A -85,B 0,C 180,E1 -20544.629,E2 -20544.629} C_VEL
LIN {X 0,Y 251.999,Z 352.957,A -85,B 0,C 180,E1 -20547.033,E2 -20547.033} C_VEL
LIN {X 0,Y 256.39,Z 359.065,A -85,B 0,C 180,E1 -20549.226,E2 -20549.226} C_VEL
LIN {X 0,Y 260.172,Z 365.181,A -85,B 0,C 180,E1 -20550.993,E2 -20550.993} C_VEL
LIN {X 0,Y 265.336,Z 374.323,A -85,B 0,C 180,E1 -20553.232,E2 -20553.232} C_VEL
LIN {X 0,Y 271.587,Z 386.342,A -85,B 0,C 180,E1 -20555.715,E2 -20555.715} C_VEL
LIN {X 0,Y 277.381,Z 398.785,A -85,B 0,C 180,E1 -20557.852,E2 -20557.852} C_VEL
LIN {X 0,Y 275.328,Z 430.563,A -85,B 0,C 180,E1 -20558.617,E2 -20558.617} C_VEL
LIN {X 0,Y 270.113,Z 508.787,A -85,B 0,C 180,E1 -20560.517,E2 -20560.517} C_VEL
LIN {X 0,Y 268.128,Z 524.552,A -85,B 0,C 180,E1 -20561.083,E2 -20561.083} C_VEL
LIN {X 0,Y 265.206,Z 540.476,A -85,B 0,C 180,E1 -20561.853,E2 -20561.853} C_VEL
LIN {X 0,Y 261.804,Z 555.566,A -85,B 0,C 180,E1 -20562.846,E2 -20562.846} C_VEL
LIN {X 0,Y 257.411,Z 571.51,A -85,B 0,C 180,E1 -20564.218,E2 -20564.218} C_VEL
LIN {X 0,Y 252.438,Z 586.75,A -85,B 0,C 180,E1 -20565.893,E2 -20565.893} C_VEL
LIN {X 0,Y 247.748,Z 599.52,A -85,B 0,C 180,E1 -20567.639,E2 -20567.639} C_VEL
LIN {X 0,Y 242.377,Z 612.662,A -85,B 0,C 180,E1 -20569.822,E2 -20569.822} C_VEL
LIN {X 0,Y 237.471,Z 623.888,A -85,B 0,C 180,E1 -20572.114,E2 -20572.114} C_VEL
LIN {X 0,Y 232.262,Z 635.085,A -85,B 0,C 180,E1 -20574.906,E2 -20574.906} C_VEL
LIN {X 0,Y 227.61,Z 644.702,A -85,B 0,C 180,E1 -20577.817,E2 -20577.817} C_VEL
LIN {X 0,Y 223.012,Z 654.061,A -85,B 0,C 180,E1 -20581.277,E2 -20581.277} C_VEL
LIN {X 0,Y 218.79,Z 662.745,A -85,B 0,C 180,E1 -20585.318,E2 -20585.318} C_VEL
LIN {X 0,Y 215.291,Z 670.444,A -85,B 0,C 180,E1 -20589.955,E2 -20589.955} C_VEL
LIN {X 0,Y 213.415,Z 675.235,A -85,B 0,C 180,E1 -20593.745,E2 -20593.745} C_VEL
LIN {X 0,Y 212.365,Z 678.156,A -85,B 0,C 180,E1 -20596.606,E2 -20596.606} C_VEL
LIN {X 0,Y 211.603,Z 681.125,A -85,B 0,C 180,E1 -20600.441,E2 -20600.441} C_VEL
LIN {X 0,Y 211.381,Z 683.089,A -85,B 0,C 180,E1 -20604.276,E2 -20604.276} C_VEL
LIN {X 0,Y 211.451,Z 684.063,A -85,B 0,C 180,E1 -20608.095,E2 -20608.095} C_VEL
LIN {X 0,Y 211.545,Z 684.22,A -85,B 0,C 180,E1 -20610,E2 -20610} C_VEL
LIN {X 0,Y 211.391,Z 683.587,A -85,B 0,C 180,E1 -20614.145,E2 -20614.145} C_VEL
LIN {X 0,Y 211.433,Z 682.24,A -85,B 0,C 180,E1 -20617.641,E2 -20617.641} C_VEL
LIN {X 0,Y 211.884,Z 679.721,A -85,B 0,C 180,E1 -20621.479,E2 -20621.479} C_VEL
LIN {X 0,Y 213.007,Z 676.27,A -85,B 0,C 180,E1 -20625.305,E2 -20625.305} C_VEL
LIN {X 0,Y 214.741,Z 671.656,A -85,B 0,C 180,E1 -20629.104,E2 -20629.104} C_VEL
LIN {X 0,Y 217.228,Z 665.948,A -85,B 0,C 180,E1 -20632.845,E2 -20632.845} C_VEL
LIN {X 0,Y 220.564,Z 659.001,A -85,B 0,C 180,E1 -20636.493,E2 -20636.493} C_VEL
LIN {X 0,Y 224.637,Z 650.596,A -85,B 0,C 180,E1 -20640.038,E2 -20640.038} C_VEL
LIN {X 0,Y 229.626,Z 640.618,A -85,B 0,C 180,E1 -20643.429,E2 -20643.429} C_VEL
LIN {X 0,Y 234.32,Z 630.522,A -85,B 0,C 180,E1 -20646.271,E2 -20646.271} C_VEL
LIN {X 0,Y 239.833,Z 618.321,A -85,B 0,C 180,E1 -20649.052,E2 -20649.052} C_VEL
LIN {X 0,Y 244.564,Z 607.214,A -85,B 0,C 180,E1 -20651.098,E2 -20651.098} C_VEL
LIN {X 0,Y 249.579,Z 594.414,A -85,B 0,C 180,E1 -20653.068,E2 -20653.068} C_VEL
LIN {X 0,Y 254.385,Z 580.716,A -85,B 0,C 180,E1 -20654.789,E2 -20654.789} C_VEL
LIN {X 0,Y 258.939,Z 565.812,A -85,B 0,C 180,E1 -20656.273,E2 -20656.273} C_VEL
LIN {X 0,Y 262.857,Z 550.618,A -85,B 0,C 180,E1 -20657.471,E2 -20657.471} C_VEL
LIN {X 0,Y 266.017,Z 535.729,A -85,B 0,C 180,E1 -20658.383,E2 -20658.383} C_VEL
LIN {X 0,Y 268.761,Z 519.219,A -85,B 0,C 180,E1 -20659.114,E2 -20659.114} C_VEL
LIN {X 0,Y 270.4,Z 503.077,A -85,B 0,C 180,E1 -20659.621,E2 -20659.621} C_VEL
LIN {X 0,Y 277.254,Z 398.781,A -85,B 0,C 180,E1 -20662.116,E2 -20662.116} C_VEL
LIN {X 0,Y 271.231,Z 385.812,A -85,B 0,C 180,E1 -20664.338,E2 -20664.338} C_VEL
LIN {X 0,Y 265.702,Z 375.173,A -85,B 0,C 180,E1 -20666.524,E2 -20666.524} C_VEL
LIN {X 0,Y 261.086,Z 366.943,A -85,B 0,C 180,E1 -20668.494,E2 -20668.494} C_VEL
LIN {X 0,Y 256.497,Z 359.228,A -85,B 0,C 180,E1 -20670.618,E2 -20670.618} C_VEL
LIN {X 0,Y 252.643,Z 353.934,A -85,B 0,C 180,E1 -20672.51,E2 -20672.51} C_VEL
LIN {X 0,Y 250.163,Z 350.534,A -85,B 0,C 180,E1 -20673.825,E2 -20673.825} C_VEL
LIN {X 0,Y 247.305,Z 346.675,A -85,B 0,C 180,E1 -20675.453,E2 -20675.453} C_VEL
LIN {X 0,Y 243.783,Z 342.071,A -85,B 0,C 180,E1 -20677.655,E2 -20677.655} C_VEL
LIN {X 0,Y 240.993,Z 338.873,A -85,B 0,C 180,E1 -20679.572,E2 -20679.572} C_VEL
LIN {X 0,Y 239.897,Z 337.189,A -85,B 0,C 180,E1 -20680.423,E2 -20680.423} C_VEL
LIN {X 0,Y 237.134,Z 334.315,A -85,B 0,C 180,E1 -20682.649,E2 -20682.649} C_VEL
LIN {X 0,Y 235.862,Z 332.004,A -85,B 0,C 180,E1 -20683.896,E2 -20683.896} C_VEL
LIN {X 0,Y 232.993,Z 329.62,A -85,B 0,C 180,E1 -20686.814,E2 -20686.814} C_VEL
LIN {X 0,Y 231.253,Z 326.349,A -85,B 0,C 180,E1 -20689.272,E2 -20689.272} C_VEL
LIN {X 0,Y 227.513,Z 322.502,A -85,B 0,C 180,E1 -20700,E2 -20700} C_VEL
LIN {X 0,Y 227.615,Z 323.318,A -85,B 0,C 180,E1 -20702.655,E2 -20702.655} C_VEL
LIN {X 0,Y 231.461,Z 326.662,A -85,B 0,C 180,E1 -20711.494,E2 -20711.494} C_VEL
LIN {X 0,Y 232.771,Z 329.288,A -85,B 0,C 180,E1 -20713.366,E2 -20713.366} C_VEL
LIN {X 0,Y 235.119,Z 331.564,A -85,B 0,C 180,E1 -20715.882,E2 -20715.882} C_VEL
LIN {X 0,Y 236.024,Z 332.341,A -85,B 0,C 180,E1 -20716.729,E2 -20716.729} C_VEL
LIN {X 0,Y 238.433,Z 335.965,A -85,B 0,C 180,E1 -20718.919,E2 -20718.919} C_VEL
LIN {X 0,Y 240.346,Z 337.736,A -85,B 0,C 180,E1 -20720.375,E2 -20720.375} C_VEL
LIN {X 0,Y 243.014,Z 341.392,A -85,B 0,C 180,E1 -20722.308,E2 -20722.308} C_VEL
LIN {X 0,Y 244.516,Z 343.012,A -85,B 0,C 180,E1 -20723.279,E2 -20723.279} C_VEL
LIN {X 0,Y 247.646,Z 346.987,A -85,B 0,C 180,E1 -20725.194,E2 -20725.194} C_VEL
LIN {X 0,Y 252.673,Z 353.971,A -85,B 0,C 180,E1 -20727.961,E2 -20727.961} C_VEL
LIN {X 0,Y 257.661,Z 360.844,A -85,B 0,C 180,E1 -20730.378,E2 -20730.378} C_VEL
LIN {X 0,Y 264.612,Z 371.323,A -85,B 0,C 180,E1 -20733.389,E2 -20733.389} C_VEL
LIN {X 0,Y 271.312,Z 382.494,A -85,B 0,C 180,E1 -20735.994,E2 -20735.994} C_VEL
LIN {X 0,Y 277.468,Z 393.576,A -85,B 0,C 180,E1 -20738.183,E2 -20738.183} C_VEL
LIN {X 0,Y 270.665,Z 496.993,A -85,B 0,C 180,E1 -20740.689,E2 -20740.689} C_VEL
LIN {X 0,Y 268.795,Z 513.067,A -85,B 0,C 180,E1 -20741.262,E2 -20741.262} C_VEL
LIN {X 0,Y 266.186,Z 528.78,A -85,B 0,C 180,E1 -20742.049,E2 -20742.049} C_VEL
LIN {X 0,Y 262.944,Z 544.331,A -85,B 0,C 180,E1 -20743.113,E2 -20743.113} C_VEL
LIN {X 0,Y 259.146,Z 558.546,A -85,B 0,C 180,E1 -20744.334,E2 -20744.334} C_VEL
LIN {X 0,Y 254.498,Z 573.674,A -85,B 0,C 180,E1 -20745.974,E2 -20745.974} C_VEL
LIN {X 0,Y 249.815,Z 587.182,A -85,B 0,C 180,E1 -20747.804,E2 -20747.804} C_VEL
LIN {X 0,Y 245.415,Z 598.335,A -85,B 0,C 180,E1 -20749.616,E2 -20749.616} C_VEL
LIN {X 0,Y 240.061,Z 610.772,A -85,B 0,C 180,E1 -20752.063,E2 -20752.063} C_VEL
LIN {X 0,Y 234.83,Z 622.17,A -85,B 0,C 180,E1 -20754.823,E2 -20754.823} C_VEL
LIN {X 0,Y 230.094,Z 631.93,A -85,B 0,C 180,E1 -20757.689,E2 -20757.689} C_VEL
LIN {X 0,Y 225.598,Z 640.778,A -85,B 0,C 180,E1 -20760.89,E2 -20760.89} C_VEL
LIN {X 0,Y 221.307,Z 649.128,A -85,B 0,C 180,E1 -20764.614,E2 -20764.614} C_VEL
LIN {X 0,Y 218.036,Z 655.657,A -85,B 0,C 180,E1 -20768.242,E2 -20768.242} C_VEL
LIN {X 0,Y 215.482,Z 660.935,A -85,B 0,C 180,E1 -20771.95,E2 -20771.95} C_VEL
LIN {X 0,Y 214.024,Z 664.193,A -85,B 0,C 180,E1 -20774.77,E2 -20774.77} C_VEL
LIN {X 0,Y 212.68,Z 667.538,A -85,B 0,C 180,E1 -20778.564,E2 -20778.564} C_VEL
LIN {X 0,Y 211.884,Z 669.967,A -85,B 0,C 180,E1 -20782.376,E2 -20782.376} C_VEL
LIN {X 0,Y 211.564,Z 671.339,A -85,B 0,C 180,E1 -20786.19,E2 -20786.19} C_VEL
LIN {X 0,Y 211.576,Z 671.865,A -85,B 0,C 180,E1 -20790,E2 -20790} C_VEL
LIN {X 0,Y 211.563,Z 671.374,A -85,B 0,C 180,E1 -20793.809,E2 -20793.809} C_VEL
LIN {X 0,Y 211.884,Z 670.035,A -85,B 0,C 180,E1 -20797.624,E2 -20797.624} C_VEL
LIN {X 0,Y 212.668,Z 667.64,A -85,B 0,C 180,E1 -20801.436,E2 -20801.436} C_VEL
LIN {X 0,Y 213.993,Z 664.336,A -85,B 0,C 180,E1 -20805.232,E2 -20805.232} C_VEL
LIN {X 0,Y 216.558,Z 658.862,A -85,B 0,C 180,E1 -20809.755,E2 -20809.755} C_VEL
LIN {X 0,Y 219.517,Z 652.767,A -85,B 0,C 180,E1 -20813.59,E2 -20813.59} C_VEL
LIN {X 0,Y 223.228,Z 645.663,A -85,B 0,C 180,E1 -20817.162,E2 -20817.162} C_VEL
LIN {X 0,Y 227.488,Z 637.161,A -85,B 0,C 180,E1 -20820.647,E2 -20820.647} C_VEL
LIN {X 0,Y 232.648,Z 626.935,A -85,B 0,C 180,E1 -20823.977,E2 -20823.977} C_VEL
LIN {X 0,Y 238.192,Z 615.252,A -85,B 0,C 180,E1 -20827.044,E2 -20827.044} C_VEL
LIN {X 0,Y 243.196,Z 603.886,A -85,B 0,C 180,E1 -20829.476,E2 -20829.476} C_VEL
LIN {X 0,Y 247.916,Z 592.49,A -85,B 0,C 180,E1 -20831.501,E2 -20831.501} C_VEL
LIN {X 0,Y 252.852,Z 579.051,A -85,B 0,C 180,E1 -20833.465,E2 -20833.465} C_VEL
LIN {X 0,Y 257.018,Z 566.186,A -85,B 0,C 180,E1 -20835.006,E2 -20835.006} C_VEL
LIN {X 0,Y 261.022,Z 552.374,A -85,B 0,C 180,E1 -20836.353,E2 -20836.353} C_VEL
LIN {X 0,Y 264.833,Z 536.551,A -85,B 0,C 180,E1 -20837.567,E2 -20837.567} C_VEL
LIN {X 0,Y 267.703,Z 520.839,A -85,B 0,C 180,E1 -20838.506,E2 -20838.506} C_VEL
LIN {X 0,Y 270.069,Z 504.231,A -85,B 0,C 180,E1 -20839.196,E2 -20839.196} C_VEL
LIN {X 0,Y 271.725,Z 484.167,A -85,B 0,C 180,E1 -20839.764,E2 -20839.764} C_VEL
LIN {X 0,Y 277.561,Z 393.589,A -85,B 0,C 180,E1 -20841.948,E2 -20841.948} C_VEL
LIN {X 0,Y 270.514,Z 380.978,A -85,B 0,C 180,E1 -20844.474,E2 -20844.474} C_VEL
LIN {X 0,Y 264.005,Z 370.318,A -85,B 0,C 180,E1 -20847.039,E2 -20847.039} C_VEL
LIN {X 0,Y 257.303,Z 360.196,A -85,B 0,C 180,E1 -20849.987,E2 -20849.987} C_VEL
LIN {X 0,Y 250.886,Z 351.345,A -85,B 0,C 180,E1 -20853.201,E2 -20853.201} C_VEL
LIN {X 0,Y 247.197,Z 346.51,A -85,B 0,C 180,E1 -20855.29,E2 -20855.29} C_VEL
LIN {X 0,Y 243.881,Z 342.147,A -85,B 0,C 180,E1 -20857.385,E2 -20857.385} C_VEL
LIN {X 0,Y 241.012,Z 338.795,A -85,B 0,C 180,E1 -20859.378,E2 -20859.378} C_VEL
LIN {X 0,Y 239.957,Z 337.185,A -85,B 0,C 180,E1 -20860.205,E2 -20860.205} C_VEL
LIN {X 0,Y 237.326,Z 334.575,A -85,B 0,C 180,E1 -20862.33,E2 -20862.33} C_VEL
LIN {X 0,Y 235.741,Z 331.887,A -85,B 0,C 180,E1 -20863.886,E2 -20863.886} C_VEL
LIN {X 0,Y 232.947,Z 329.577,A -85,B 0,C 180,E1 -20866.811,E2 -20866.811} C_VEL
LIN {X 0,Y 231.424,Z 326.439,A -85,B 0,C 180,E1 -20869.058,E2 -20869.058} C_VEL
LIN {X 0,Y 227.776,Z 323.152,A -85,B 0,C 180,E1 -20879.116,E2 -20879.116} C_VEL
LIN {X 0,Y 227.841,Z 323.361,A -85,B 0,C 180,E1 -20881.572,E2 -20881.572} C_VEL
LIN {X 0,Y 227.949,Z 324.52,A -85,B 0,C 180,E1 -20883.029,E2 -20883.029} C_VEL
LIN {X 0,Y 228.829,Z 331.834,A -85,B 0,C 180,E1 -20887.652,E2 -20887.652} C_VEL
LIN {X 0,Y 229.553,Z 332.974,A -85,B 0,C 180,E1 -20889.089,E2 -20889.089} C_VEL
LIN {X 0,Y 230.341,Z 333.557,A -85,B 0,C 180,E1 -20890.32,E2 -20890.32} C_VEL
LIN {X 0,Y 232.059,Z 336.823,A -85,B 0,C 180,E1 -20892.85,E2 -20892.85} C_VEL
LIN {X 0,Y 234.681,Z 339.165,A -85,B 0,C 180,E1 -20895.636,E2 -20895.636} C_VEL
LIN {X 0,Y 237.018,Z 342.684,A -85,B 0,C 180,E1 -20897.861,E2 -20897.861} C_VEL
LIN {X 0,Y 238.79,Z 344.442,A -85,B 0,C 180,E1 -20899.28,E2 -20899.28} C_VEL
LIN {X 0,Y 241.527,Z 348.186,A -85,B 0,C 180,E1 -20901.34,E2 -20901.34} C_VEL
LIN {X 0,Y 242.823,Z 349.644,A -85,B 0,C 180,E1 -20902.214,E2 -20902.214} C_VEL
LIN {X 0,Y 246.719,Z 354.922,A -85,B 0,C 180,E1 -20904.676,E2 -20904.676} C_VEL
LIN {X 0,Y 250.033,Z 359.527,A -85,B 0,C 180,E1 -20906.557,E2 -20906.557} C_VEL
LIN {X 0,Y 254.688,Z 366.102,A -85,B 0,C 180,E1 -20908.941,E2 -20908.941} C_VEL
LIN {X 0,Y 260.586,Z 376.576,A -85,B 0,C 180,E1 -20911.729,E2 -20911.729} C_VEL
LIN {X 0,Y 265.781,Z 386.566,A -85,B 0,C 180,E1 -20913.959,E2 -20913.959} C_VEL
LIN {X 0,Y 271.343,Z 398.083,A -85,B 0,C 180,E1 -20916.161,E2 -20916.161} C_VEL
LIN {X 0,Y 272.924,Z 402.042,A -85,B 0,C 180,E1 -20916.78,E2 -20916.78} C_VEL
LIN {X 0,Y 265.495,Z 509.347,A -85,B 0,C 180,E1 -20919.374,E2 -20919.374} C_VEL
LIN {X 0,Y 263.215,Z 526.066,A -85,B 0,C 180,E1 -20919.98,E2 -20919.98} C_VEL
LIN {X 0,Y 260.026,Z 542.531,A -85,B 0,C 180,E1 -20920.819,E2 -20920.819} C_VEL
LIN {X 0,Y 256.165,Z 558.348,A -85,B 0,C 180,E1 -20921.911,E2 -20921.911} C_VEL
LIN {X 0,Y 251.964,Z 572.958,A -85,B 0,C 180,E1 -20923.223,E2 -20923.223} C_VEL
LIN {X 0,Y 246.864,Z 587.974,A -85,B 0,C 180,E1 -20924.914,E2 -20924.914} C_VEL
LIN {X 0,Y 241.638,Z 601.502,A -85,B 0,C 180,E1 -20926.836,E2 -20926.836} C_VEL
LIN {X 0,Y 236.027,Z 614.415,A -85,B 0,C 180,E1 -20929.075,E2 -20929.075} C_VEL
LIN {X 0,Y 231.029,Z 625.406,A -85,B 0,C 180,E1 -20931.42,E2 -20931.42} C_VEL
LIN {X 0,Y 225.704,Z 636.399,A -85,B 0,C 180,E1 -20934.289,E2 -20934.289} C_VEL
LIN {X 0,Y 220.87,Z 645.734,A -85,B 0,C 180,E1 -20937.253,E2 -20937.253} C_VEL
LIN {X 0,Y 216.17,Z 654.87,A -85,B 0,C 180,E1 -20940.813,E2 -20940.813} C_VEL
LIN {X 0,Y 212.254,Z 662.535,A -85,B 0,C 180,E1 -20944.504,E2 -20944.504} C_VEL
LIN {X 0,Y 208.528,Z 670.235,A -85,B 0,C 180,E1 -20949.275,E2 -20949.275} C_VEL
LIN {X 0,Y 206.524,Z 675.026,A -85,B 0,C 180,E1 -20953.187,E2 -20953.187} C_VEL
LIN {X 0,Y 205.379,Z 677.947,A -85,B 0,C 180,E1 -20956.141,E2 -20956.141} C_VEL
LIN {X 0,Y 204.55,Z 680.916,A -85,B 0,C 180,E1 -20960.108,E2 -20960.108} C_VEL
LIN {X 0,Y 204.286,Z 682.881,A -85,B 0,C 180,E1 -20964.076,E2 -20964.076} C_VEL
LIN {X 0,Y 204.353,Z 683.855,A -85,B 0,C 180,E1 -20968.029,E2 -20968.029} C_VEL
LIN {X 0,Y 204.463,Z 684.013,A -85,B 0,C 180,E1 -20970,E2 -20970} C_VEL
LIN {X 0,Y 204.319,Z 683.44,A -85,B 0,C 180,E1 -20974.045,E2 -20974.045} C_VEL
LIN {X 0,Y 204.366,Z 682.031,A -85,B 0,C 180,E1 -20977.907,E2 -20977.907} C_VEL
LIN {X 0,Y 204.853,Z 679.511,A -85,B 0,C 180,E1 -20981.879,E2 -20981.879} C_VEL
LIN {X 0,Y 206.084,Z 676.059,A -85,B 0,C 180,E1 -20985.832,E2 -20985.832} C_VEL
LIN {X 0,Y 207.936,Z 671.444,A -85,B 0,C 180,E1 -20989.754,E2 -20989.754} C_VEL
LIN {X 0,Y 210.593,Z 665.736,A -85,B 0,C 180,E1 -20993.607,E2 -20993.607} C_VEL
LIN {X 0,Y 214.141,Z 658.789,A -85,B 0,C 180,E1 -20997.353,E2 -20997.353} C_VEL
LIN {X 0,Y 218.427,Z 650.384,A -85,B 0,C 180,E1 -21000.984,E2 -21000.984} C_VEL
LIN {X 0,Y 223.617,Z 640.405,A -85,B 0,C 180,E1 -21004.452,E2 -21004.452} C_VEL
LIN {X 0,Y 227.878,Z 631.729,A -85,B 0,C 180,E1 -21006.97,E2 -21006.97} C_VEL
LIN {X 0,Y 233.449,Z 619.904,A -85,B 0,C 180,E1 -21009.772,E2 -21009.772} C_VEL
LIN {X 0,Y 238.74,Z 608.075,A -85,B 0,C 180,E1 -21012.044,E2 -21012.044} C_VEL
LIN {X 0,Y 244.409,Z 594.201,A -85,B 0,C 180,E1 -21014.211,E2 -21014.211} C_VEL
LIN {X 0,Y 249.376,Z 580.504,A -85,B 0,C 180,E1 -21015.943,E2 -21015.943} C_VEL
LIN {X 0,Y 254.055,Z 565.598,A -85,B 0,C 180,E1 -21017.437,E2 -21017.437} C_VEL
LIN {X 0,Y 258.075,Z 550.402,A -85,B 0,C 180,E1 -21018.641,E2 -21018.641} C_VEL
LIN {X 0,Y 261.499,Z 534.626,A -85,B 0,C 180,E1 -21019.596,E2 -21019.596} C_VEL
LIN {X 0,Y 264.333,Z 517.977,A -85,B 0,C 180,E1 -21020.305,E2 -21020.305} C_VEL
LIN {X 0,Y 265.958,Z 501.492,A -85,B 0,C 180,E1 -21020.827,E2 -21020.827} C_VEL
LIN {X 0,Y 272.763,Z 401.585,A -85,B 0,C 180,E1 -21023.215,E2 -21023.215} C_VEL
LIN {X 0,Y 267.174,Z 389.502,A -85,B 0,C 180,E1 -21025.388,E2 -21025.388} C_VEL
LIN {X 0,Y 261.697,Z 378.735,A -85,B 0,C 180,E1 -21027.684,E2 -21027.684} C_VEL
LIN {X 0,Y 256.56,Z 369.491,A -85,B 0,C 180,E1 -21030.029,E2 -21030.029} C_VEL
LIN {X 0,Y 253.472,Z 364.473,A -85,B 0,C 180,E1 -21031.54,E2 -21031.54} C_VEL
LIN {X 0,Y 248.41,Z 357.229,A -85,B 0,C 180,E1 -21034.216,E2 -21034.216} C_VEL
LIN {X 0,Y 244.857,Z 352.51,A -85,B 0,C 180,E1 -21036.307,E2 -21036.307} C_VEL
LIN {X 0,Y 241.916,Z 348.573,A -85,B 0,C 180,E1 -21038.234,E2 -21038.234} C_VEL
LIN {X 0,Y 239.005,Z 344.9,A -85,B 0,C 180,E1 -21040.347,E2 -21040.347} C_VEL
LIN {X 0,Y 238.246,Z 343.823,A -85,B 0,C 180,E1 -21040.954,E2 -21040.954} C_VEL
LIN {X 0,Y 235.465,Z 340.663,A -85,B 0,C 180,E1 -21043.316,E2 -21043.316} C_VEL
LIN {X 0,Y 234.454,Z 338.818,A -85,B 0,C 180,E1 -21044.349,E2 -21044.349} C_VEL
LIN {X 0,Y 231.521,Z 336.109,A -85,B 0,C 180,E1 -21047.509,E2 -21047.509} C_VEL
LIN {X 0,Y 230.234,Z 333.428,A -85,B 0,C 180,E1 -21049.447,E2 -21049.447} C_VEL
LIN {X 0,Y 226.647,Z 329.559,A -85,B 0,C 180,E1 -21060,E2 -21060} C_VEL
LIN {X 0,Y 226.804,Z 330.596,A -85,B 0,C 180,E1 -21063.109,E2 -21063.109} C_VEL
LIN {X 0,Y 230.293,Z 333.555,A -85,B 0,C 180,E1 -21071.107,E2 -21071.107} C_VEL
LIN {X 0,Y 231.767,Z 336.436,A -85,B 0,C 180,E1 -21073.257,E2 -21073.257} C_VEL
LIN {X 0,Y 234.602,Z 339.091,A -85,B 0,C 180,E1 -21076.263,E2 -21076.263} C_VEL
LIN {X 0,Y 236.929,Z 342.619,A -85,B 0,C 180,E1 -21078.455,E2 -21078.455} C_VEL
LIN {X 0,Y 238.752,Z 344.428,A -85,B 0,C 180,E1 -21079.899,E2 -21079.899} C_VEL
LIN {X 0,Y 241.591,Z 348.259,A -85,B 0,C 180,E1 -21082.006,E2 -21082.006} C_VEL
LIN {X 0,Y 242.821,Z 349.722,A -85,B 0,C 180,E1 -21082.832,E2 -21082.832} C_VEL
LIN {X 0,Y 246.384,Z 354.545,A -85,B 0,C 180,E1 -21085.075,E2 -21085.075} C_VEL
LIN {X 0,Y 250.078,Z 359.679,A -85,B 0,C 180,E1 -21087.165,E2 -21087.165} C_VEL
LIN {X 0,Y 254.958,Z 366.485,A -85,B 0,C 180,E1 -21089.634,E2 -21089.634} C_VEL
LIN {X 0,Y 261.775,Z 377.067,A -85,B 0,C 180,E1 -21092.715,E2 -21092.715} C_VEL
LIN {X 0,Y 268.204,Z 388.029,A -85,B 0,C 180,E1 -21095.315,E2 -21095.315} C_VEL
LIN {X 0,Y 272.936,Z 396.653,A -85,B 0,C 180,E1 -21097.078,E2 -21097.078} C_VEL
LIN {X 0,Y 266.025,Z 498.035,A -85,B 0,C 180,E1 -21099.553,E2 -21099.553} C_VEL
LIN {X 0,Y 264.044,Z 514.2,A -85,B 0,C 180,E1 -21100.147,E2 -21100.147} C_VEL
LIN {X 0,Y 261.216,Z 530.292,A -85,B 0,C 180,E1 -21100.973,E2 -21100.973} C_VEL
LIN {X 0,Y 257.881,Z 545.571,A -85,B 0,C 180,E1 -21102.044,E2 -21102.044} C_VEL
LIN {X 0,Y 253.745,Z 560.518,A -85,B 0,C 180,E1 -21103.361,E2 -21103.361} C_VEL
LIN {X 0,Y 249.303,Z 574.24,A -85,B 0,C 180,E1 -21104.88,E2 -21104.88} C_VEL
LIN {X 0,Y 244.133,Z 588.561,A -85,B 0,C 180,E1 -21106.867,E2 -21106.867} C_VEL
LIN {X 0,Y 239.594,Z 599.61,A -85,B 0,C 180,E1 -21108.701,E2 -21108.701} C_VEL
LIN {X 0,Y 234.471,Z 610.983,A -85,B 0,C 180,E1 -21110.991,E2 -21110.991} C_VEL
LIN {X 0,Y 229.034,Z 622.381,A -85,B 0,C 180,E1 -21113.794,E2 -21113.794} C_VEL
LIN {X 0,Y 224.076,Z 632.141,A -85,B 0,C 180,E1 -21116.71,E2 -21116.71} C_VEL
LIN {X 0,Y 219.145,Z 641.417,A -85,B 0,C 180,E1 -21120.151,E2 -21120.151} C_VEL
LIN {X 0,Y 214.864,Z 649.338,A -85,B 0,C 180,E1 -21123.796,E2 -21123.796} C_VEL
LIN {X 0,Y 211.387,Z 655.868,A -85,B 0,C 180,E1 -21127.521,E2 -21127.521} C_VEL
LIN {X 0,Y 208.688,Z 661.145,A -85,B 0,C 180,E1 -21131.341,E2 -21131.341} C_VEL
LIN {X 0,Y 207.152,Z 664.402,A -85,B 0,C 180,E1 -21134.252,E2 -21134.252} C_VEL
LIN {X 0,Y 205.698,Z 667.747,A -85,B 0,C 180,E1 -21138.171,E2 -21138.171} C_VEL
LIN {X 0,Y 204.845,Z 670.174,A -85,B 0,C 180,E1 -21142.112,E2 -21142.112} C_VEL
LIN {X 0,Y 204.474,Z 671.547,A -85,B 0,C 180,E1 -21146.058,E2 -21146.058} C_VEL
LIN {X 0,Y 204.494,Z 672.072,A -85,B 0,C 180,E1 -21150,E2 -21150} C_VEL
LIN {X 0,Y 204.531,Z 671.377,A -85,B 0,C 180,E1 -21154.805,E2 -21154.805} C_VEL
LIN {X 0,Y 204.844,Z 670.242,A -85,B 0,C 180,E1 -21157.888,E2 -21157.888} C_VEL
LIN {X 0,Y 205.685,Z 667.848,A -85,B 0,C 180,E1 -21161.83,E2 -21161.83} C_VEL
LIN {X 0,Y 207.118,Z 664.544,A -85,B 0,C 180,E1 -21165.751,E2 -21165.751} C_VEL
LIN {X 0,Y 209.653,Z 659.376,A -85,B 0,C 180,E1 -21170.179,E2 -21170.179} C_VEL
LIN {X 0,Y 212.968,Z 652.975,A -85,B 0,C 180,E1 -21174.362,E2 -21174.362} C_VEL
LIN {X 0,Y 216.886,Z 645.87,A -85,B 0,C 180,E1 -21178.025,E2 -21178.025} C_VEL
LIN {X 0,Y 221.365,Z 637.368,A -85,B 0,C 180,E1 -21181.59,E2 -21181.59} C_VEL
LIN {X 0,Y 226.76,Z 627.141,A -85,B 0,C 180,E1 -21184.985,E2 -21184.985} C_VEL
LIN {X 0,Y 232.29,Z 615.927,A -85,B 0,C 180,E1 -21187.992,E2 -21187.992} C_VEL
LIN {X 0,Y 237.741,Z 604.091,A -85,B 0,C 180,E1 -21190.568,E2 -21190.568} C_VEL
LIN {X 0,Y 242.64,Z 592.693,A -85,B 0,C 180,E1 -21192.613,E2 -21192.613} C_VEL
LIN {X 0,Y 247.583,Z 579.646,A -85,B 0,C 180,E1 -21194.546,E2 -21194.546} C_VEL
LIN {X 0,Y 252.092,Z 566.232,A -85,B 0,C 180,E1 -21196.166,E2 -21196.166} C_VEL
LIN {X 0,Y 256.177,Z 552.575,A -85,B 0,C 180,E1 -21197.501,E2 -21197.501} C_VEL
LIN {X 0,Y 260.091,Z 536.751,A -85,B 0,C 180,E1 -21198.723,E2 -21198.723} C_VEL
LIN {X 0,Y 263.055,Z 521.036,A -85,B 0,C 180,E1 -21199.664,E2 -21199.664} C_VEL
LIN {X 0,Y 265.526,Z 504.052,A -85,B 0,C 180,E1 -21200.369,E2 -21200.369} C_VEL
LIN {X 0,Y 267.27,Z 483.208,A -85,B 0,C 180,E1 -21200.954,E2 -21200.954} C_VEL
LIN {X 0,Y 273.105,Z 396.782,A -85,B 0,C 180,E1 -21203.03,E2 -21203.03} C_VEL
LIN {X 0,Y 266.315,Z 384.602,A -85,B 0,C 180,E1 -21205.598,E2 -21205.598} C_VEL
LIN {X 0,Y 260.56,Z 375.082,A -85,B 0,C 180,E1 -21207.99,E2 -21207.99} C_VEL
LIN {X 0,Y 254.65,Z 365.986,A -85,B 0,C 180,E1 -21210.715,E2 -21210.715} C_VEL
LIN {X 0,Y 248.847,Z 357.728,A -85,B 0,C 180,E1 -21213.74,E2 -21213.74} C_VEL
LIN {X 0,Y 245.183,Z 352.836,A -85,B 0,C 180,E1 -21215.891,E2 -21215.891} C_VEL
LIN {X 0,Y 242.067,Z 348.658,A -85,B 0,C 180,E1 -21217.936,E2 -21217.936} C_VEL
LIN {X 0,Y 239.143,Z 344.997,A -85,B 0,C 180,E1 -21220.068,E2 -21220.068} C_VEL
LIN {X 0,Y 238.351,Z 343.884,A -85,B 0,C 180,E1 -21220.706,E2 -21220.706} C_VEL
LIN {X 0,Y 235.674,Z 340.943,A -85,B 0,C 180,E1 -21222.983,E2 -21222.983} C_VEL
LIN {X 0,Y 234.35,Z 338.677,A -85,B 0,C 180,E1 -21224.341,E2 -21224.341} C_VEL
LIN {X 0,Y 231.578,Z 336.164,A -85,B 0,C 180,E1 -21227.401,E2 -21227.401} C_VEL
LIN {X 0,Y 230.27,Z 333.337,A -85,B 0,C 180,E1 -21229.448,E2 -21229.448} C_VEL
LIN {X 0,Y 226.91,Z 330.21,A -85,B 0,C 180,E1 -21239.112,E2 -21239.112} C_VEL
LIN {X 0,Y 226.988,Z 330.513,A -85,B 0,C 180,E1 -21241.774,E2 -21241.774} C_VEL
LIN {X 0,Y 229.553,Z 332.974,A -85,B 0,C 180,E1 -21249.089,E2 -21249.089} C_VEL
LIN {X 0,Y 229.969,Z 333.892,A -85,B 0,C 180,E1 -21249.867,E2 -21249.867} C_VEL
LIN {X 0,Y 230.346,Z 336.578,A -85,B 0,C 180,E1 -21250.821,E2 -21250.821} C_VEL
LIN {X 0,Y 231.055,Z 342.944,A -85,B 0,C 180,E1 -21252.599,E2 -21252.599} C_VEL
LIN {X 0,Y 231.708,Z 344.547,A -85,B 0,C 180,E1 -21253.5,E2 -21253.5} C_VEL
LIN {X 0,Y 233.29,Z 345.927,A -85,B 0,C 180,E1 -21255.172,E2 -21255.172} C_VEL
LIN {X 0,Y 235.857,Z 349.72,A -85,B 0,C 180,E1 -21257.672,E2 -21257.672} C_VEL
LIN {X 0,Y 237.22,Z 351.12,A -85,B 0,C 180,E1 -21258.795,E2 -21258.795} C_VEL
LIN {X 0,Y 240.092,Z 354.99,A -85,B 0,C 180,E1 -21261.013,E2 -21261.013} C_VEL
LIN {X 0,Y 241.484,Z 356.885,A -85,B 0,C 180,E1 -21261.996,E2 -21261.996} C_VEL
LIN {X 0,Y 244.715,Z 361.251,A -85,B 0,C 180,E1 -21264.09,E2 -21264.09} C_VEL
LIN {X 0,Y 248.298,Z 366.375,A -85,B 0,C 180,E1 -21266.191,E2 -21266.191} C_VEL
LIN {X 0,Y 252.405,Z 372.363,A -85,B 0,C 180,E1 -21268.365,E2 -21268.365} C_VEL
LIN {X 0,Y 257.674,Z 382.055,A -85,B 0,C 180,E1 -21270.965,E2 -21270.965} C_VEL
LIN {X 0,Y 262.616,Z 391.833,A -85,B 0,C 180,E1 -21273.184,E2 -21273.184} C_VEL
LIN {X 0,Y 268.162,Z 403.644,A -85,B 0,C 180,E1 -21275.478,E2 -21275.478} C_VEL
LIN {X 0,Y 268.517,Z 404.575,A -85,B 0,C 180,E1 -21275.625,E2 -21275.625} C_VEL
LIN {X 0,Y 261.096,Z 508.385,A -85,B 0,C 180,E1 -21278.142,E2 -21278.142} C_VEL
LIN {X 0,Y 258.836,Z 525.194,A -85,B 0,C 180,E1 -21278.752,E2 -21278.752} C_VEL
LIN {X 0,Y 255.865,Z 540.372,A -85,B 0,C 180,E1 -21279.496,E2 -21279.496} C_VEL
LIN {X 0,Y 252.355,Z 555.163,A -85,B 0,C 180,E1 -21280.48,E2 -21280.48} C_VEL
LIN {X 0,Y 247.688,Z 571.105,A -85,B 0,C 180,E1 -21281.856,E2 -21281.856} C_VEL
LIN {X 0,Y 242.395,Z 586.342,A -85,B 0,C 180,E1 -21283.544,E2 -21283.544} C_VEL
LIN {X 0,Y 237.016,Z 599.936,A -85,B 0,C 180,E1 -21285.436,E2 -21285.436} C_VEL
LIN {X 0,Y 231.585,Z 612.248,A -85,B 0,C 180,E1 -21287.529,E2 -21287.529} C_VEL
LIN {X 0,Y 226.299,Z 623.474,A -85,B 0,C 180,E1 -21289.879,E2 -21289.879} C_VEL
LIN {X 0,Y 220.445,Z 635.001,A -85,B 0,C 180,E1 -21292.846,E2 -21292.846} C_VEL
LIN {X 0,Y 215.565,Z 644.285,A -85,B 0,C 180,E1 -21295.779,E2 -21295.779} C_VEL
LIN {X 0,Y 210.49,Z 653.643,A -85,B 0,C 180,E1 -21299.391,E2 -21299.391} C_VEL
LIN {X 0,Y 206.676,Z 660.498,A -85,B 0,C 180,E1 -21302.673,E2 -21302.673} C_VEL
LIN {X 0,Y 203.205,Z 667.146,A -85,B 0,C 180,E1 -21306.564,E2 -21306.564} C_VEL
LIN {X 0,Y 200.544,Z 672.68,A -85,B 0,C 180,E1 -21310.66,E2 -21310.66} C_VEL
LIN {X 0,Y 199.189,Z 675.899,A -85,B 0,C 180,E1 -21313.605,E2 -21313.605} C_VEL
LIN {X 0,Y 197.833,Z 679.337,A -85,B 0,C 180,E1 -21317.693,E2 -21317.693} C_VEL
LIN {X 0,Y 197.289,Z 681.847,A -85,B 0,C 180,E1 -21321.808,E2 -21321.808} C_VEL
LIN {X 0,Y 197.24,Z 683.314,A -85,B 0,C 180,E1 -21326.096,E2 -21326.096} C_VEL
LIN {X 0,Y 197.363,Z 683.806,A -85,B 0,C 180,E1 -21330,E2 -21330} C_VEL
LIN {X 0,Y 197.243,Z 683.258,A -85,B 0,C 180,E1 -21334.087,E2 -21334.087} C_VEL
LIN {X 0,Y 197.289,Z 681.822,A -85,B 0,C 180,E1 -21338.192,E2 -21338.192} C_VEL
LIN {X 0,Y 197.832,Z 679.3,A -85,B 0,C 180,E1 -21342.307,E2 -21342.307} C_VEL
LIN {X 0,Y 199.186,Z 675.849,A -85,B 0,C 180,E1 -21346.396,E2 -21346.396} C_VEL
LIN {X 0,Y 201.17,Z 671.233,A -85,B 0,C 180,E1 -21350.448,E2 -21350.448} C_VEL
LIN {X 0,Y 204.002,Z 665.524,A -85,B 0,C 180,E1 -21354.419,E2 -21354.419} C_VEL
LIN {X 0,Y 208.078,Z 657.962,A -85,B 0,C 180,E1 -21358.579,E2 -21358.579} C_VEL
LIN {X 0,Y 212.905,Z 649.045,A -85,B 0,C 180,E1 -21362.44,E2 -21362.44} C_VEL
LIN {X 0,Y 217.669,Z 640.191,A -85,B 0,C 180,E1 -21365.533,E2 -21365.533} C_VEL
LIN {X 0,Y 222.167,Z 631.516,A -85,B 0,C 180,E1 -21368.087,E2 -21368.087} C_VEL
LIN {X 0,Y 227.981,Z 619.691,A -85,B 0,C 180,E1 -21370.925,E2 -21370.925} C_VEL
LIN {X 0,Y 233.484,Z 607.863,A -85,B 0,C 180,E1 -21373.219,E2 -21373.219} C_VEL
LIN {X 0,Y 238.821,Z 595.285,A -85,B 0,C 180,E1 -21375.23,E2 -21375.23} C_VEL
LIN {X 0,Y 244.467,Z 580.291,A -85,B 0,C 180,E1 -21377.145,E2 -21377.145} C_VEL
LIN {X 0,Y 249.288,Z 565.385,A -85,B 0,C 180,E1 -21378.644,E2 -21378.644} C_VEL
LIN {X 0,Y 253.429,Z 550.188,A -85,B 0,C 180,E1 -21379.849,E2 -21379.849} C_VEL
LIN {X 0,Y 257.056,Z 533.844,A -85,B 0,C 180,E1 -21380.831,E2 -21380.831} C_VEL
LIN {X 0,Y 259.867,Z 517.668,A -85,B 0,C 180,E1 -21381.512,E2 -21381.512} C_VEL
LIN {X 0,Y 261.528,Z 501.266,A -85,B 0,C 180,E1 -21382.034,E2 -21382.034} C_VEL
LIN {X 0,Y 268.356,Z 404.456,A -85,B 0,C 180,E1 -21384.353,E2 -21384.353} C_VEL
LIN {X 0,Y 263.267,Z 393.33,A -85,B 0,C 180,E1 -21386.445,E2 -21386.445} C_VEL
LIN {X 0,Y 258.198,Z 383.233,A -85,B 0,C 180,E1 -21388.687,E2 -21388.687} C_VEL
LIN {X 0,Y 254.007,Z 375.397,A -85,B 0,C 180,E1 -21390.7,E2 -21390.7} C_VEL
LIN {X 0,Y 251.051,Z 370.455,A -85,B 0,C 180,E1 -21392.207,E2 -21392.207} C_VEL
LIN {X 0,Y 246.074,Z 363.235,A -85,B 0,C 180,E1 -21394.949,E2 -21394.949} C_VEL
LIN {X 0,Y 242.772,Z 358.694,A -85,B 0,C 180,E1 -21396.984,E2 -21396.984} C_VEL
LIN {X 0,Y 240.015,Z 354.943,A -85,B 0,C 180,E1 -21398.868,E2 -21398.868} C_VEL
LIN {X 0,Y 236.494,Z 350.303,A -85,B 0,C 180,E1 -21401.594,E2 -21401.594} C_VEL
LIN {X 0,Y 233.85,Z 347.041,A -85,B 0,C 180,E1 -21403.97,E2 -21403.97} C_VEL
LIN {X 0,Y 232.927,Z 345.533,A -85,B 0,C 180,E1 -21404.939,E2 -21404.939} C_VEL
LIN {X 0,Y 230.164,Z 342.692,A -85,B 0,C 180,E1 -21408.106,E2 -21408.106} C_VEL
LIN {X 0,Y 228.968,Z 340.224,A -85,B 0,C 180,E1 -21410.008,E2 -21410.008} C_VEL
LIN {X 0,Y 225.78,Z 336.618,A -85,B 0,C 180,E1 -21420,E2 -21420} C_VEL
LIN {X 0,Y 229.074,Z 340.307,A -85,B 0,C 180,E1 -21430.608,E2 -21430.608} C_VEL
LIN {X 0,Y 230.644,Z 343.371,A -85,B 0,C 180,E1 -21432.987,E2 -21432.987} C_VEL
LIN {X 0,Y 233.272,Z 345.965,A -85,B 0,C 180,E1 -21435.872,E2 -21435.872} C_VEL
LIN {X 0,Y 235.617,Z 349.49,A -85,B 0,C 180,E1 -21438.14,E2 -21438.14} C_VEL
LIN {X 0,Y 237.235,Z 351.226,A -85,B 0,C 180,E1 -21439.468,E2 -21439.468} C_VEL
LIN {X 0,Y 240.231,Z 355.151,A -85,B 0,C 180,E1 -21441.737,E2 -21441.737} C_VEL
LIN {X 0,Y 244.45,Z 360.998,A -85,B 0,C 180,E1 -21444.533,E2 -21444.533} C_VEL
LIN {X 0,Y 248.44,Z 366.644,A -85,B 0,C 180,E1 -21446.855,E2 -21446.855} C_VEL
LIN {X 0,Y 253.871,Z 374.65,A -85,B 0,C 180,E1 -21449.659,E2 -21449.659} C_VEL
LIN {X 0,Y 259.932,Z 384.447,A -85,B 0,C 180,E1 -21452.448,E2 -21452.448} C_VEL
LIN {X 0,Y 266.099,Z 395.278,A -85,B 0,C 180,E1 -21455.002,E2 -21455.002} C_VEL
LIN {X 0,Y 268.541,Z 399.841,A -85,B 0,C 180,E1 -21455.951,E2 -21455.951} C_VEL
LIN {X 0,Y 261.549,Z 498.611,A -85,B 0,C 180,E1 -21458.368,E2 -21458.368} C_VEL
LIN {X 0,Y 259.386,Z 515.334,A -85,B 0,C 180,E1 -21458.988,E2 -21458.988} C_VEL
